   1:  PR[GP1:91,1] = PR[GP1:90,1] + 125.067;
   1:  PR[GP1:91,2] = PR[GP1:90,2] + 105.676;
   1:L PR[91] 10mm/sec FINE;
   1:  PR[GP1:91,1] = PR[GP1:90,1] + 125.211;
   1:  PR[GP1:91,2] = PR[GP1:90,2] + 108.371;
   1:L PR[91] 10mm/sec FINE;
   1:  PR[GP1:91,1] = PR[GP1:90,1] + 124.783;
   1:  PR[GP1:91,2] = PR[GP1:90,2] + 111.876;
   1:L PR[91] 10mm/sec FINE;
   1:  PR[GP1:91,1] = PR[GP1:90,1] + 123.660;
   1:  PR[GP1:91,2] = PR[GP1:90,2] + 115.178;
   1:L PR[91] 10mm/sec FINE;
   1:  PR[GP1:91,1] = PR[GP1:90,1] + 121.852;
   1:  PR[GP1:91,2] = PR[GP1:90,2] + 118.170;
   1:L PR[91] 10mm/sec FINE;
   1:  PR[GP1:91,1] = PR[GP1:90,1] + 119.446;
   1:  PR[GP1:91,2] = PR[GP1:90,2] + 120.740;
   1:L PR[91] 10mm/sec FINE;
   1:  PR[GP1:91,1] = PR[GP1:90,1] + 116.594;
   1:  PR[GP1:91,2] = PR[GP1:90,2] + 122.770;
   1:L PR[91] 10mm/sec FINE;
   1:  PR[GP1:91,1] = PR[GP1:90,1] + 113.357;
   1:  PR[GP1:91,2] = PR[GP1:90,2] + 124.215;
   1:L PR[91] 10mm/sec FINE;
   1:  PR[GP1:91,1] = PR[GP1:90,1] + 109.836;
   1:  PR[GP1:91,2] = PR[GP1:90,2] + 125.035;
   1:L PR[91] 10mm/sec FINE;
   1:  PR[GP1:91,1] = PR[GP1:90,1] + 106.255;
   1:  PR[GP1:91,2] = PR[GP1:90,2] + 125.172;
   1:L PR[91] 10mm/sec FINE;
   1:  PR[GP1:91,1] = PR[GP1:90,1] + 102.748;
   1:  PR[GP1:91,2] = PR[GP1:90,2] + 124.631;
   1:L PR[91] 10mm/sec FINE;
   1:  PR[GP1:91,1] = PR[GP1:90,1] + 99.339;
   1:  PR[GP1:91,2] = PR[GP1:90,2] + 123.456;
   1:L PR[91] 10mm/sec FINE;
   1:  PR[GP1:91,1] = PR[GP1:90,1] + 97.309;
   1:  PR[GP1:91,2] = PR[GP1:90,2] + 122.401;
   1:L PR[91] 10mm/sec FINE;
   1:  PR[GP1:91,1] = PR[GP1:90,1] + 96.953;
   1:  PR[GP1:91,2] = PR[GP1:90,2] + 122.201;
   1:L PR[91] 10mm/sec FINE;
   1:  PR[GP1:91,1] = PR[GP1:90,1] + 95.813;
   1:  PR[GP1:91,2] = PR[GP1:90,2] + 121.862;
   1:L PR[91] 10mm/sec FINE;
   1:  PR[GP1:91,1] = PR[GP1:90,1] + 94.847;
   1:  PR[GP1:91,2] = PR[GP1:90,2] + 122.067;
   1:L PR[91] 10mm/sec FINE;
   1:  PR[GP1:91,1] = PR[GP1:90,1] + 93.928;
   1:  PR[GP1:91,2] = PR[GP1:90,2] + 122.476;
   1:L PR[91] 10mm/sec FINE;
   1:  PR[GP1:91,1] = PR[GP1:90,1] + 93.286;
   1:  PR[GP1:91,2] = PR[GP1:90,2] + 122.743;
   1:L PR[91] 10mm/sec FINE;
   1:  PR[GP1:91,1] = PR[GP1:90,1] + 90.578;
   1:  PR[GP1:91,2] = PR[GP1:90,2] + 123.691;
   1:L PR[91] 10mm/sec FINE;
   1:  PR[GP1:91,1] = PR[GP1:90,1] + 89.346;
   1:  PR[GP1:91,2] = PR[GP1:90,2] + 123.990;
   1:L PR[91] 10mm/sec FINE;
   1:  PR[GP1:91,1] = PR[GP1:90,1] + 87.282;
   1:  PR[GP1:91,2] = PR[GP1:90,2] + 124.465;
   1:L PR[91] 10mm/sec FINE;
   1:  PR[GP1:91,1] = PR[GP1:90,1] + 86.381;
   1:  PR[GP1:91,2] = PR[GP1:90,2] + 124.569;
   1:L PR[91] 10mm/sec FINE;
   1:  PR[GP1:91,1] = PR[GP1:90,1] + 83.107;
   1:  PR[GP1:91,2] = PR[GP1:90,2] + 124.845;
   1:L PR[91] 10mm/sec FINE;
   1:  PR[GP1:91,1] = PR[GP1:90,1] + 82.927;
   1:  PR[GP1:91,2] = PR[GP1:90,2] + 124.844;
   1:L PR[91] 10mm/sec FINE;
   1:  PR[GP1:91,1] = PR[GP1:90,1] + 79.793;
   1:  PR[GP1:91,2] = PR[GP1:90,2] + 124.596;
   1:L PR[91] 10mm/sec FINE;
   1:  PR[GP1:91,1] = PR[GP1:90,1] + 78.215;
   1:  PR[GP1:91,2] = PR[GP1:90,2] + 124.296;
   1:L PR[91] 10mm/sec FINE;
   1:  PR[GP1:91,1] = PR[GP1:90,1] + 76.415;
   1:  PR[GP1:91,2] = PR[GP1:90,2] + 123.822;
   1:L PR[91] 10mm/sec FINE;
   1:  PR[GP1:91,1] = PR[GP1:90,1] + 73.897;
   1:  PR[GP1:91,2] = PR[GP1:90,2] + 122.815;
   1:L PR[91] 10mm/sec FINE;
   1:  PR[GP1:91,1] = PR[GP1:90,1] + 73.134;
   1:  PR[GP1:91,2] = PR[GP1:90,2] + 122.451;
   1:L PR[91] 10mm/sec FINE;
   1:  PR[GP1:91,1] = PR[GP1:90,1] + 70.131;
   1:  PR[GP1:91,2] = PR[GP1:90,2] + 120.456;
   1:L PR[91] 10mm/sec FINE;
   1:  PR[GP1:91,1] = PR[GP1:90,1] + 69.386;
   1:  PR[GP1:91,2] = PR[GP1:90,2] + 119.681;
   1:L PR[91] 10mm/sec FINE;
   1:  PR[GP1:91,1] = PR[GP1:90,1] + 67.649;
   1:  PR[GP1:91,2] = PR[GP1:90,2] + 117.796;
   1:L PR[91] 10mm/sec FINE;
   1:  PR[GP1:91,1] = PR[GP1:90,1] + 65.840;
   1:  PR[GP1:91,2] = PR[GP1:90,2] + 114.671;
   1:L PR[91] 10mm/sec FINE;
   1:  PR[GP1:91,1] = PR[GP1:90,1] + 64.732;
   1:  PR[GP1:91,2] = PR[GP1:90,2] + 111.266;
   1:L PR[91] 10mm/sec FINE;
   1:  PR[GP1:91,1] = PR[GP1:90,1] + 64.492;
   1:  PR[GP1:91,2] = PR[GP1:90,2] + 107.656;
   1:L PR[91] 10mm/sec FINE;
   1:  PR[GP1:91,1] = PR[GP1:90,1] + 65.074;
   1:  PR[GP1:91,2] = PR[GP1:90,2] + 104.024;
   1:L PR[91] 10mm/sec FINE;
   1:  PR[GP1:91,1] = PR[GP1:90,1] + 65.085;
   1:  PR[GP1:91,2] = PR[GP1:90,2] + 103.970;
   1:L PR[91] 10mm/sec FINE;
   1:  PR[GP1:91,1] = PR[GP1:90,1] + 66.507;
   1:  PR[GP1:91,2] = PR[GP1:90,2] + 100.470;
   1:L PR[91] 10mm/sec FINE;
   1:  PR[GP1:91,1] = PR[GP1:90,1] + 66.955;
   1:  PR[GP1:91,2] = PR[GP1:90,2] + 99.803;
   1:L PR[91] 10mm/sec FINE;
   1:  PR[GP1:91,1] = PR[GP1:90,1] + 68.693;
   1:  PR[GP1:91,2] = PR[GP1:90,2] + 97.301;
   1:L PR[91] 10mm/sec FINE;
   1:  PR[GP1:91,1] = PR[GP1:90,1] + 70.114;
   1:  PR[GP1:91,2] = PR[GP1:90,2] + 95.877;
   1:L PR[91] 10mm/sec FINE;
   1:  PR[GP1:91,1] = PR[GP1:90,1] + 71.437;
   1:  PR[GP1:91,2] = PR[GP1:90,2] + 94.608;
   1:L PR[91] 10mm/sec FINE;
   1:  PR[GP1:91,1] = PR[GP1:90,1] + 73.564;
   1:  PR[GP1:91,2] = PR[GP1:90,2] + 93.370;
   1:  PR[GP1:91,3] = PR[GP1:90,3] + 32.900;
   1:L PR[91] 10mm/sec FINE;
   1:  PR[GP1:91,1] = PR[GP1:90,1] + 75.182;
   1:  PR[GP1:91,2] = PR[GP1:90,2] + 92.299;
   1:L PR[91] 10mm/sec FINE;
   1:  PR[GP1:91,1] = PR[GP1:90,1] + 76.014;
   1:  PR[GP1:91,2] = PR[GP1:90,2] + 91.905;
   1:L PR[91] 10mm/sec FINE;
   1:  PR[GP1:91,1] = PR[GP1:90,1] + 78.652;
   1:  PR[GP1:91,2] = PR[GP1:90,2] + 90.708;
   1:L PR[91] 10mm/sec FINE;
   1:  PR[GP1:91,1] = PR[GP1:90,1] + 81.260;
   1:  PR[GP1:91,2] = PR[GP1:90,2] + 89.873;
   1:L PR[91] 10mm/sec FINE;
   1:  PR[GP1:91,1] = PR[GP1:90,1] + 81.725;
   1:  PR[GP1:91,2] = PR[GP1:90,2] + 89.744;
   1:L PR[91] 10mm/sec FINE;
   1:  PR[GP1:91,1] = PR[GP1:90,1] + 82.381;
   1:  PR[GP1:91,2] = PR[GP1:90,2] + 89.624;
   1:L PR[91] 10mm/sec FINE;
   1:  PR[GP1:91,1] = PR[GP1:90,1] + 85.201;
   1:  PR[GP1:91,2] = PR[GP1:90,2] + 89.020;
   1:L PR[91] 10mm/sec FINE;
   1:  PR[GP1:91,1] = PR[GP1:90,1] + 87.810;
   1:  PR[GP1:91,2] = PR[GP1:90,2] + 88.790;
   1:L PR[91] 10mm/sec FINE;
   1:  PR[GP1:91,1] = PR[GP1:90,1] + 89.579;
   1:  PR[GP1:91,2] = PR[GP1:90,2] + 88.697;
   1:L PR[91] 10mm/sec FINE;
   1:  PR[GP1:91,1] = PR[GP1:90,1] + 91.610;
   1:  PR[GP1:91,2] = PR[GP1:90,2] + 88.771;
   1:L PR[91] 10mm/sec FINE;
   1:  PR[GP1:91,1] = PR[GP1:90,1] + 94.675;
   1:  PR[GP1:91,2] = PR[GP1:90,2] + 89.210;
   1:L PR[91] 10mm/sec FINE;
   1:  PR[GP1:91,1] = PR[GP1:90,1] + 95.921;
   1:  PR[GP1:91,2] = PR[GP1:90,2] + 89.430;
   1:L PR[91] 10mm/sec FINE;
   1:  PR[GP1:91,1] = PR[GP1:90,1] + 97.181;
   1:  PR[GP1:91,2] = PR[GP1:90,2] + 89.860;
   1:L PR[91] 10mm/sec FINE;
   1:  PR[GP1:91,1] = PR[GP1:90,1] + 97.451;
   1:  PR[GP1:91,2] = PR[GP1:90,2] + 89.925;
   1:L PR[91] 10mm/sec FINE;
   1:  PR[GP1:91,1] = PR[GP1:90,1] + 98.662;
   1:  PR[GP1:91,2] = PR[GP1:90,2] + 89.766;
   1:L PR[91] 10mm/sec FINE;
   1:  PR[GP1:91,1] = PR[GP1:90,1] + 100.674;
   1:  PR[GP1:91,2] = PR[GP1:90,2] + 89.073;
   1:L PR[91] 10mm/sec FINE;
   1:  PR[GP1:91,1] = PR[GP1:90,1] + 100.904;
   1:  PR[GP1:91,2] = PR[GP1:90,2] + 88.999;
   1:L PR[91] 10mm/sec FINE;
   1:  PR[GP1:91,1] = PR[GP1:90,1] + 101.374;
   1:  PR[GP1:91,2] = PR[GP1:90,2] + 88.890;
   1:L PR[91] 10mm/sec FINE;
   1:  PR[GP1:91,1] = PR[GP1:90,1] + 103.724;
   1:  PR[GP1:91,2] = PR[GP1:90,2] + 88.477;
   1:L PR[91] 10mm/sec FINE;
   1:  PR[GP1:91,1] = PR[GP1:90,1] + 104.087;
   1:  PR[GP1:91,2] = PR[GP1:90,2] + 88.454;
   1:L PR[91] 10mm/sec FINE;
   1:  PR[GP1:91,1] = PR[GP1:90,1] + 106.621;
   1:  PR[GP1:91,2] = PR[GP1:90,2] + 88.429;
   1:L PR[91] 10mm/sec FINE;
   1:  PR[GP1:91,1] = PR[GP1:90,1] + 109.525;
   1:  PR[GP1:91,2] = PR[GP1:90,2] + 88.858;
   1:L PR[91] 10mm/sec FINE;
   1:  PR[GP1:91,1] = PR[GP1:90,1] + 112.350;
   1:  PR[GP1:91,2] = PR[GP1:90,2] + 89.744;
   1:L PR[91] 10mm/sec FINE;
   1:  PR[GP1:91,1] = PR[GP1:90,1] + 115.027;
   1:  PR[GP1:91,2] = PR[GP1:90,2] + 91.077;
   1:L PR[91] 10mm/sec FINE;
   1:  PR[GP1:91,1] = PR[GP1:90,1] + 117.480;
   1:  PR[GP1:91,2] = PR[GP1:90,2] + 92.827;
   1:L PR[91] 10mm/sec FINE;
   1:  PR[GP1:91,1] = PR[GP1:90,1] + 119.096;
   1:  PR[GP1:91,2] = PR[GP1:90,2] + 94.413;
   1:L PR[91] 10mm/sec FINE;
   1:  PR[GP1:91,1] = PR[GP1:90,1] + 119.702;
   1:  PR[GP1:91,2] = PR[GP1:90,2] + 94.984;
   1:L PR[91] 10mm/sec FINE;
   1:  PR[GP1:91,1] = PR[GP1:90,1] + 121.111;
   1:  PR[GP1:91,2] = PR[GP1:90,2] + 96.735;
   1:L PR[91] 10mm/sec FINE;
   1:  PR[GP1:91,1] = PR[GP1:90,1] + 121.662;
   1:  PR[GP1:91,2] = PR[GP1:90,2] + 97.494;
   1:L PR[91] 10mm/sec FINE;
   1:  PR[GP1:91,1] = PR[GP1:90,1] + 122.375;
   1:  PR[GP1:91,2] = PR[GP1:90,2] + 98.721;
   1:L PR[91] 10mm/sec FINE;
   1:  PR[GP1:91,1] = PR[GP1:90,1] + 123.132;
   1:  PR[GP1:91,2] = PR[GP1:90,2] + 100.157;
   1:L PR[91] 10mm/sec FINE;
   1:  PR[GP1:91,1] = PR[GP1:90,1] + 123.382;
   1:  PR[GP1:91,2] = PR[GP1:90,2] + 100.787;
   1:L PR[91] 10mm/sec FINE;
   1:  PR[GP1:91,1] = PR[GP1:90,1] + 124.131;
   1:  PR[GP1:91,2] = PR[GP1:90,2] + 102.876;
   1:L PR[91] 10mm/sec FINE;
   1:  PR[GP1:91,1] = PR[GP1:90,1] + 124.717;
   1:  PR[GP1:91,2] = PR[GP1:90,2] + 105.523;
   1:L PR[91] 10mm/sec FINE;
   1:  PR[GP1:91,1] = PR[GP1:90,1] + 124.859;
   1:  PR[GP1:91,2] = PR[GP1:90,2] + 108.206;
   1:L PR[91] 10mm/sec FINE;
   1:  PR[GP1:91,1] = PR[GP1:90,1] + 124.427;
   1:  PR[GP1:91,2] = PR[GP1:90,2] + 111.723;
   1:L PR[91] 10mm/sec FINE;
   1:  PR[GP1:91,1] = PR[GP1:90,1] + 123.294;
   1:  PR[GP1:91,2] = PR[GP1:90,2] + 115.038;
   1:L PR[91] 10mm/sec FINE;
   1:  PR[GP1:91,1] = PR[GP1:90,1] + 121.502;
   1:  PR[GP1:91,2] = PR[GP1:90,2] + 118.026;
   1:L PR[91] 10mm/sec FINE;
   1:  PR[GP1:91,1] = PR[GP1:90,1] + 119.130;
   1:  PR[GP1:91,2] = PR[GP1:90,2] + 120.582;
   1:L PR[91] 10mm/sec FINE;
   1:  PR[GP1:91,1] = PR[GP1:90,1] + 118.062;
   1:  PR[GP1:91,2] = PR[GP1:90,2] + 121.345;
   1:L PR[91] 10mm/sec FINE;
   1:  PR[GP1:91,1] = PR[GP1:90,1] + 116.272;
   1:  PR[GP1:91,2] = PR[GP1:90,2] + 122.619;
   1:L PR[91] 10mm/sec FINE;
   1:  PR[GP1:91,1] = PR[GP1:90,1] + 113.025;
   1:  PR[GP1:91,2] = PR[GP1:90,2] + 124.072;
   1:L PR[91] 10mm/sec FINE;
   1:  PR[GP1:91,1] = PR[GP1:90,1] + 109.576;
   1:  PR[GP1:91,2] = PR[GP1:90,2] + 124.872;
   1:L PR[91] 10mm/sec FINE;
   1:  PR[GP1:91,1] = PR[GP1:90,1] + 106.003;
   1:  PR[GP1:91,2] = PR[GP1:90,2] + 125.012;
   1:L PR[91] 10mm/sec FINE;
   1:  PR[GP1:91,1] = PR[GP1:90,1] + 104.565;
   1:  PR[GP1:91,2] = PR[GP1:90,2] + 124.806;
   1:L PR[91] 10mm/sec FINE;
   1:  PR[GP1:91,1] = PR[GP1:90,1] + 102.475;
   1:  PR[GP1:91,2] = PR[GP1:90,2] + 124.481;
   1:L PR[91] 10mm/sec FINE;
   1:  PR[GP1:91,1] = PR[GP1:90,1] + 99.066;
   1:  PR[GP1:91,2] = PR[GP1:90,2] + 123.311;
   1:L PR[91] 10mm/sec FINE;
   1:  PR[GP1:91,1] = PR[GP1:90,1] + 97.099;
   1:  PR[GP1:91,2] = PR[GP1:90,2] + 122.284;
   1:L PR[91] 10mm/sec FINE;
   1:  PR[GP1:91,1] = PR[GP1:90,1] + 96.627;
   1:  PR[GP1:91,2] = PR[GP1:90,2] + 122.161;
   1:L PR[91] 10mm/sec FINE;
   1:  PR[GP1:91,1] = PR[GP1:90,1] + 95.962;
   1:  PR[GP1:91,2] = PR[GP1:90,2] + 121.960;
   1:L PR[91] 10mm/sec FINE;
   1:  PR[GP1:91,1] = PR[GP1:90,1] + 95.071;
   1:  PR[GP1:91,2] = PR[GP1:90,2] + 122.159;
   1:L PR[91] 10mm/sec FINE;
   1:  PR[GP1:91,1] = PR[GP1:90,1] + 93.990;
   1:  PR[GP1:91,2] = PR[GP1:90,2] + 122.603;
   1:L PR[91] 10mm/sec FINE;
   1:  PR[GP1:91,1] = PR[GP1:90,1] + 91.198;
   1:  PR[GP1:91,2] = PR[GP1:90,2] + 123.560;
   1:L PR[91] 10mm/sec FINE;
   1:  PR[GP1:91,1] = PR[GP1:90,1] + 88.055;
   1:  PR[GP1:91,2] = PR[GP1:90,2] + 124.289;
   1:L PR[91] 10mm/sec FINE;
   1:  PR[GP1:91,1] = PR[GP1:90,1] + 86.606;
   1:  PR[GP1:91,2] = PR[GP1:90,2] + 124.457;
   1:L PR[91] 10mm/sec FINE;
   1:  PR[GP1:91,1] = PR[GP1:90,1] + 83.984;
   1:  PR[GP1:91,2] = PR[GP1:90,2] + 124.674;
   1:L PR[91] 10mm/sec FINE;
   1:  PR[GP1:91,1] = PR[GP1:90,1] + 83.485;
   1:  PR[GP1:91,2] = PR[GP1:90,2] + 124.677;
   1:L PR[91] 10mm/sec FINE;
   1:  PR[GP1:91,1] = PR[GP1:90,1] + 80.051;
   1:  PR[GP1:91,2] = PR[GP1:90,2] + 124.408;
   1:L PR[91] 10mm/sec FINE;
   1:  PR[GP1:91,1] = PR[GP1:90,1] + 79.265;
   1:  PR[GP1:91,2] = PR[GP1:90,2] + 124.259;
   1:L PR[91] 10mm/sec FINE;
   1:  PR[GP1:91,1] = PR[GP1:90,1] + 76.736;
   1:  PR[GP1:91,2] = PR[GP1:90,2] + 123.592;
   1:L PR[91] 10mm/sec FINE;
   1:  PR[GP1:91,1] = PR[GP1:90,1] + 74.918;
   1:  PR[GP1:91,2] = PR[GP1:90,2] + 122.866;
   1:L PR[91] 10mm/sec FINE;
   1:  PR[GP1:91,1] = PR[GP1:90,1] + 73.515;
   1:  PR[GP1:91,2] = PR[GP1:90,2] + 122.198;
   1:L PR[91] 10mm/sec FINE;
   1:  PR[GP1:91,1] = PR[GP1:90,1] + 71.197;
   1:  PR[GP1:91,2] = PR[GP1:90,2] + 120.664;
   1:L PR[91] 10mm/sec FINE;
   1:  PR[GP1:91,1] = PR[GP1:90,1] + 70.574;
   1:  PR[GP1:91,2] = PR[GP1:90,2] + 120.197;
   1:L PR[91] 10mm/sec FINE;
   1:  PR[GP1:91,1] = PR[GP1:90,1] + 68.301;
   1:  PR[GP1:91,2] = PR[GP1:90,2] + 117.833;
   1:L PR[91] 10mm/sec FINE;
   1:  PR[GP1:91,1] = PR[GP1:90,1] + 68.113;
   1:  PR[GP1:91,2] = PR[GP1:90,2] + 117.615;
   1:L PR[91] 10mm/sec FINE;
   1:  PR[GP1:91,1] = PR[GP1:90,1] + 66.280;
   1:  PR[GP1:91,2] = PR[GP1:90,2] + 114.537;
   1:L PR[91] 10mm/sec FINE;
   1:  PR[GP1:91,1] = PR[GP1:90,1] + 65.163;
   1:  PR[GP1:91,2] = PR[GP1:90,2] + 111.135;
   1:L PR[91] 10mm/sec FINE;
   1:  PR[GP1:91,1] = PR[GP1:90,1] + 64.981;
   1:  PR[GP1:91,2] = PR[GP1:90,2] + 107.692;
   1:L PR[91] 10mm/sec FINE;
   1:  PR[GP1:91,1] = PR[GP1:90,1] + 64.960;
   1:  PR[GP1:91,2] = PR[GP1:90,2] + 107.499;
   1:L PR[91] 10mm/sec FINE;
   1:  PR[GP1:91,1] = PR[GP1:90,1] + 65.415;
   1:  PR[GP1:91,2] = PR[GP1:90,2] + 104.903;
   1:L PR[91] 10mm/sec FINE;
   1:  PR[GP1:91,1] = PR[GP1:90,1] + 65.548;
   1:  PR[GP1:91,2] = PR[GP1:90,2] + 104.351;
   1:L PR[91] 10mm/sec FINE;
   1:  PR[GP1:91,1] = PR[GP1:90,1] + 65.650;
   1:  PR[GP1:91,2] = PR[GP1:90,2] + 103.812;
   1:L PR[91] 10mm/sec FINE;
   1:  PR[GP1:91,1] = PR[GP1:90,1] + 67.051;
   1:  PR[GP1:91,2] = PR[GP1:90,2] + 100.343;
   1:L PR[91] 10mm/sec FINE;
   1:  PR[GP1:91,1] = PR[GP1:90,1] + 67.947;
   1:  PR[GP1:91,2] = PR[GP1:90,2] + 99.007;
   1:L PR[91] 10mm/sec FINE;
   1:  PR[GP1:91,1] = PR[GP1:90,1] + 69.205;
   1:  PR[GP1:91,2] = PR[GP1:90,2] + 97.197;
   1:L PR[91] 10mm/sec FINE;
   1:  PR[GP1:91,1] = PR[GP1:90,1] + 71.256;
   1:  PR[GP1:91,2] = PR[GP1:90,2] + 95.142;
   1:L PR[91] 10mm/sec FINE;
   1:  PR[GP1:91,1] = PR[GP1:90,1] + 71.906;
   1:  PR[GP1:91,2] = PR[GP1:90,2] + 94.518;
   1:L PR[91] 10mm/sec FINE;
   1:  PR[GP1:91,1] = PR[GP1:90,1] + 75.880;
   1:  PR[GP1:91,2] = PR[GP1:90,2] + 92.109;
   1:  PR[GP1:91,3] = PR[GP1:90,3] + 33.900;
   1:L PR[91] 10mm/sec FINE;
   1:  PR[GP1:91,1] = PR[GP1:90,1] + 77.710;
   1:  PR[GP1:91,2] = PR[GP1:90,2] + 91.243;
   1:L PR[91] 10mm/sec FINE;
   1:  PR[GP1:91,1] = PR[GP1:90,1] + 79.190;
   1:  PR[GP1:91,2] = PR[GP1:90,2] + 90.572;
   1:L PR[91] 10mm/sec FINE;
   1:  PR[GP1:91,1] = PR[GP1:90,1] + 81.284;
   1:  PR[GP1:91,2] = PR[GP1:90,2] + 89.901;
   1:L PR[91] 10mm/sec FINE;
   1:  PR[GP1:91,1] = PR[GP1:90,1] + 82.269;
   1:  PR[GP1:91,2] = PR[GP1:90,2] + 89.559;
   1:L PR[91] 10mm/sec FINE;
   1:  PR[GP1:91,1] = PR[GP1:90,1] + 86.037;
   1:  PR[GP1:91,2] = PR[GP1:90,2] + 88.743;
   1:L PR[91] 10mm/sec FINE;
   1:  PR[GP1:91,1] = PR[GP1:90,1] + 88.313;
   1:  PR[GP1:91,2] = PR[GP1:90,2] + 88.542;
   1:L PR[91] 10mm/sec FINE;
   1:  PR[GP1:91,1] = PR[GP1:90,1] + 90.636;
   1:  PR[GP1:91,2] = PR[GP1:90,2] + 88.420;
   1:L PR[91] 10mm/sec FINE;
   1:  PR[GP1:91,1] = PR[GP1:90,1] + 92.273;
   1:  PR[GP1:91,2] = PR[GP1:90,2] + 88.479;
   1:L PR[91] 10mm/sec FINE;
   1:  PR[GP1:91,1] = PR[GP1:90,1] + 95.963;
   1:  PR[GP1:91,2] = PR[GP1:90,2] + 89.008;
   1:L PR[91] 10mm/sec FINE;
   1:  PR[GP1:91,1] = PR[GP1:90,1] + 96.765;
   1:  PR[GP1:91,2] = PR[GP1:90,2] + 89.149;
   1:L PR[91] 10mm/sec FINE;
   1:  PR[GP1:91,1] = PR[GP1:90,1] + 97.566;
   1:  PR[GP1:91,2] = PR[GP1:90,2] + 89.421;
   1:L PR[91] 10mm/sec FINE;
   1:  PR[GP1:91,1] = PR[GP1:90,1] + 97.747;
   1:  PR[GP1:91,2] = PR[GP1:90,2] + 89.464;
   1:L PR[91] 10mm/sec FINE;
   1:  PR[GP1:91,1] = PR[GP1:90,1] + 98.964;
   1:  PR[GP1:91,2] = PR[GP1:90,2] + 89.336;
   1:L PR[91] 10mm/sec FINE;
   1:  PR[GP1:91,1] = PR[GP1:90,1] + 100.640;
   1:  PR[GP1:91,2] = PR[GP1:90,2] + 88.779;
   1:L PR[91] 10mm/sec FINE;
   1:  PR[GP1:91,1] = PR[GP1:90,1] + 101.756;
   1:  PR[GP1:91,2] = PR[GP1:90,2] + 88.520;
   1:L PR[91] 10mm/sec FINE;
   1:  PR[GP1:91,1] = PR[GP1:90,1] + 103.448;
   1:  PR[GP1:91,2] = PR[GP1:90,2] + 88.222;
   1:L PR[91] 10mm/sec FINE;
   1:  PR[GP1:91,1] = PR[GP1:90,1] + 104.526;
   1:  PR[GP1:91,2] = PR[GP1:90,2] + 88.154;
   1:L PR[91] 10mm/sec FINE;
   1:  PR[GP1:91,1] = PR[GP1:90,1] + 106.342;
   1:  PR[GP1:91,2] = PR[GP1:90,2] + 88.137;
   1:L PR[91] 10mm/sec FINE;
   1:  PR[GP1:91,1] = PR[GP1:90,1] + 107.253;
   1:  PR[GP1:91,2] = PR[GP1:90,2] + 88.230;
   1:L PR[91] 10mm/sec FINE;
   1:  PR[GP1:91,1] = PR[GP1:90,1] + 109.250;
   1:  PR[GP1:91,2] = PR[GP1:90,2] + 88.541;
   1:L PR[91] 10mm/sec FINE;
   1:  PR[GP1:91,1] = PR[GP1:90,1] + 109.859;
   1:  PR[GP1:91,2] = PR[GP1:90,2] + 88.707;
   1:L PR[91] 10mm/sec FINE;
   1:  PR[GP1:91,1] = PR[GP1:90,1] + 112.092;
   1:  PR[GP1:91,2] = PR[GP1:90,2] + 89.441;
   1:L PR[91] 10mm/sec FINE;
   1:  PR[GP1:91,1] = PR[GP1:90,1] + 112.281;
   1:  PR[GP1:91,2] = PR[GP1:90,2] + 89.527;
   1:L PR[91] 10mm/sec FINE;
   1:  PR[GP1:91,1] = PR[GP1:90,1] + 113.192;
   1:  PR[GP1:91,2] = PR[GP1:90,2] + 90.000;
   1:L PR[91] 10mm/sec FINE;
   1:  PR[GP1:91,1] = PR[GP1:90,1] + 114.777;
   1:  PR[GP1:91,2] = PR[GP1:90,2] + 90.781;
   1:L PR[91] 10mm/sec FINE;
   1:  PR[GP1:91,1] = PR[GP1:90,1] + 117.237;
   1:  PR[GP1:91,2] = PR[GP1:90,2] + 92.516;
   1:L PR[91] 10mm/sec FINE;
   1:  PR[GP1:91,1] = PR[GP1:90,1] + 119.406;
   1:  PR[GP1:91,2] = PR[GP1:90,2] + 94.623;
   1:L PR[91] 10mm/sec FINE;
   1:  PR[GP1:91,1] = PR[GP1:90,1] + 121.236;
   1:  PR[GP1:91,2] = PR[GP1:90,2] + 97.056;
   1:L PR[91] 10mm/sec FINE;
   1:  PR[GP1:91,1] = PR[GP1:90,1] + 122.420;
   1:  PR[GP1:91,2] = PR[GP1:90,2] + 99.091;
   1:L PR[91] 10mm/sec FINE;
   1:  PR[GP1:91,1] = PR[GP1:90,1] + 122.771;
   1:  PR[GP1:91,2] = PR[GP1:90,2] + 99.758;
   1:L PR[91] 10mm/sec FINE;
   1:  PR[GP1:91,1] = PR[GP1:90,1] + 123.359;
   1:  PR[GP1:91,2] = PR[GP1:90,2] + 101.242;
   1:L PR[91] 10mm/sec FINE;
   1:  PR[GP1:91,1] = PR[GP1:90,1] + 123.821;
   1:  PR[GP1:91,2] = PR[GP1:90,2] + 102.530;
   1:L PR[91] 10mm/sec FINE;
   1:  PR[GP1:91,1] = PR[GP1:90,1] + 124.030;
   1:  PR[GP1:91,2] = PR[GP1:90,2] + 103.454;
   1:L PR[91] 10mm/sec FINE;
   1:  PR[GP1:91,1] = PR[GP1:90,1] + 124.403;
   1:  PR[GP1:91,2] = PR[GP1:90,2] + 105.299;
   1:L PR[91] 10mm/sec FINE;
   1:  PR[GP1:91,1] = PR[GP1:90,1] + 124.528;
   1:  PR[GP1:91,2] = PR[GP1:90,2] + 108.026;
   1:L PR[91] 10mm/sec FINE;
   1:  PR[GP1:91,1] = PR[GP1:90,1] + 124.113;
   1:  PR[GP1:91,2] = PR[GP1:90,2] + 111.543;
   1:L PR[91] 10mm/sec FINE;
   1:  PR[GP1:91,1] = PR[GP1:90,1] + 122.985;
   1:  PR[GP1:91,2] = PR[GP1:90,2] + 114.864;
   1:L PR[91] 10mm/sec FINE;
   1:  PR[GP1:91,1] = PR[GP1:90,1] + 121.192;
   1:  PR[GP1:91,2] = PR[GP1:90,2] + 117.859;
   1:L PR[91] 10mm/sec FINE;
   1:  PR[GP1:91,1] = PR[GP1:90,1] + 118.815;
   1:  PR[GP1:91,2] = PR[GP1:90,2] + 120.424;
   1:L PR[91] 10mm/sec FINE;
   1:  PR[GP1:91,1] = PR[GP1:90,1] + 115.950;
   1:  PR[GP1:91,2] = PR[GP1:90,2] + 122.468;
   1:L PR[91] 10mm/sec FINE;
   1:  PR[GP1:91,1] = PR[GP1:90,1] + 112.721;
   1:  PR[GP1:91,2] = PR[GP1:90,2] + 123.919;
   1:L PR[91] 10mm/sec FINE;
   1:  PR[GP1:91,1] = PR[GP1:90,1] + 109.316;
   1:  PR[GP1:91,2] = PR[GP1:90,2] + 124.709;
   1:L PR[91] 10mm/sec FINE;
   1:  PR[GP1:91,1] = PR[GP1:90,1] + 105.778;
   1:  PR[GP1:91,2] = PR[GP1:90,2] + 124.846;
   1:L PR[91] 10mm/sec FINE;
   1:  PR[GP1:91,1] = PR[GP1:90,1] + 102.203;
   1:  PR[GP1:91,2] = PR[GP1:90,2] + 124.331;
   1:L PR[91] 10mm/sec FINE;
   1:  PR[GP1:91,1] = PR[GP1:90,1] + 98.768;
   1:  PR[GP1:91,2] = PR[GP1:90,2] + 123.112;
   1:L PR[91] 10mm/sec FINE;
   1:  PR[GP1:91,1] = PR[GP1:90,1] + 98.344;
   1:  PR[GP1:91,2] = PR[GP1:90,2] + 122.907;
   1:L PR[91] 10mm/sec FINE;
   1:  PR[GP1:91,1] = PR[GP1:90,1] + 97.258;
   1:  PR[GP1:91,2] = PR[GP1:90,2] + 122.346;
   1:L PR[91] 10mm/sec FINE;
   1:  PR[GP1:91,1] = PR[GP1:90,1] + 96.108;
   1:  PR[GP1:91,2] = PR[GP1:90,2] + 122.055;
   1:L PR[91] 10mm/sec FINE;
   1:  PR[GP1:91,1] = PR[GP1:90,1] + 95.302;
   1:  PR[GP1:91,2] = PR[GP1:90,2] + 122.227;
   1:L PR[91] 10mm/sec FINE;
   1:  PR[GP1:91,1] = PR[GP1:90,1] + 94.695;
   1:  PR[GP1:91,2] = PR[GP1:90,2] + 122.463;
   1:L PR[91] 10mm/sec FINE;
   1:  PR[GP1:91,1] = PR[GP1:90,1] + 92.033;
   1:  PR[GP1:91,2] = PR[GP1:90,2] + 123.359;
   1:L PR[91] 10mm/sec FINE;
   1:  PR[GP1:91,1] = PR[GP1:90,1] + 88.828;
   1:  PR[GP1:91,2] = PR[GP1:90,2] + 124.113;
   1:L PR[91] 10mm/sec FINE;
   1:  PR[GP1:91,1] = PR[GP1:90,1] + 86.830;
   1:  PR[GP1:91,2] = PR[GP1:90,2] + 124.345;
   1:L PR[91] 10mm/sec FINE;
   1:  PR[GP1:91,1] = PR[GP1:90,1] + 85.063;
   1:  PR[GP1:91,2] = PR[GP1:90,2] + 124.491;
   1:L PR[91] 10mm/sec FINE;
   1:  PR[GP1:91,1] = PR[GP1:90,1] + 83.896;
   1:  PR[GP1:91,2] = PR[GP1:90,2] + 124.498;
   1:L PR[91] 10mm/sec FINE;
   1:  PR[GP1:91,1] = PR[GP1:90,1] + 80.317;
   1:  PR[GP1:91,2] = PR[GP1:90,2] + 124.221;
   1:L PR[91] 10mm/sec FINE;
   1:  PR[GP1:91,1] = PR[GP1:90,1] + 77.056;
   1:  PR[GP1:91,2] = PR[GP1:90,2] + 123.363;
   1:L PR[91] 10mm/sec FINE;
   1:  PR[GP1:91,1] = PR[GP1:90,1] + 75.938;
   1:  PR[GP1:91,2] = PR[GP1:90,2] + 122.916;
   1:L PR[91] 10mm/sec FINE;
   1:  PR[GP1:91,1] = PR[GP1:90,1] + 73.897;
   1:  PR[GP1:91,2] = PR[GP1:90,2] + 121.944;
   1:L PR[91] 10mm/sec FINE;
   1:  PR[GP1:91,1] = PR[GP1:90,1] + 72.163;
   1:  PR[GP1:91,2] = PR[GP1:90,2] + 120.797;
   1:L PR[91] 10mm/sec FINE;
   1:  PR[GP1:91,1] = PR[GP1:90,1] + 71.014;
   1:  PR[GP1:91,2] = PR[GP1:90,2] + 119.935;
   1:L PR[91] 10mm/sec FINE;
   1:  PR[GP1:91,1] = PR[GP1:90,1] + 69.191;
   1:  PR[GP1:91,2] = PR[GP1:90,2] + 118.039;
   1:L PR[91] 10mm/sec FINE;
   1:  PR[GP1:91,1] = PR[GP1:90,1] + 68.603;
   1:  PR[GP1:91,2] = PR[GP1:90,2] + 117.357;
   1:L PR[91] 10mm/sec FINE;
   1:  PR[GP1:91,1] = PR[GP1:90,1] + 67.108;
   1:  PR[GP1:91,2] = PR[GP1:90,2] + 114.852;
   1:L PR[91] 10mm/sec FINE;
   1:  PR[GP1:91,1] = PR[GP1:90,1] + 66.809;
   1:  PR[GP1:91,2] = PR[GP1:90,2] + 114.301;
   1:L PR[91] 10mm/sec FINE;
   1:  PR[GP1:91,1] = PR[GP1:90,1] + 65.875;
   1:  PR[GP1:91,2] = PR[GP1:90,2] + 111.457;
   1:L PR[91] 10mm/sec FINE;
   1:  PR[GP1:91,1] = PR[GP1:90,1] + 65.715;
   1:  PR[GP1:91,2] = PR[GP1:90,2] + 110.923;
   1:L PR[91] 10mm/sec FINE;
   1:  PR[GP1:91,1] = PR[GP1:90,1] + 65.562;
   1:  PR[GP1:91,2] = PR[GP1:90,2] + 108.031;
   1:L PR[91] 10mm/sec FINE;
   1:  PR[GP1:91,1] = PR[GP1:90,1] + 65.485;
   1:  PR[GP1:91,2] = PR[GP1:90,2] + 107.327;
   1:L PR[91] 10mm/sec FINE;
   1:  PR[GP1:91,1] = PR[GP1:90,1] + 65.756;
   1:  PR[GP1:91,2] = PR[GP1:90,2] + 105.779;
   1:L PR[91] 10mm/sec FINE;
   1:  PR[GP1:91,1] = PR[GP1:90,1] + 66.013;
   1:  PR[GP1:91,2] = PR[GP1:90,2] + 104.711;
   1:L PR[91] 10mm/sec FINE;
   1:  PR[GP1:91,1] = PR[GP1:90,1] + 66.214;
   1:  PR[GP1:91,2] = PR[GP1:90,2] + 103.656;
   1:L PR[91] 10mm/sec FINE;
   1:  PR[GP1:91,1] = PR[GP1:90,1] + 67.596;
   1:  PR[GP1:91,2] = PR[GP1:90,2] + 100.215;
   1:L PR[91] 10mm/sec FINE;
   1:  PR[GP1:91,1] = PR[GP1:90,1] + 68.940;
   1:  PR[GP1:91,2] = PR[GP1:90,2] + 98.212;
   1:L PR[91] 10mm/sec FINE;
   1:  PR[GP1:91,1] = PR[GP1:90,1] + 69.718;
   1:  PR[GP1:91,2] = PR[GP1:90,2] + 97.094;
   1:L PR[91] 10mm/sec FINE;
   1:  PR[GP1:91,1] = PR[GP1:90,1] + 72.381;
   1:  PR[GP1:91,2] = PR[GP1:90,2] + 94.425;
   1:L PR[91] 10mm/sec FINE;
   1:  PR[GP1:91,1] = PR[GP1:90,1] + 73.210;
   1:  PR[GP1:91,2] = PR[GP1:90,2] + 94.142;
   1:  PR[GP1:91,3] = PR[GP1:90,3] + 34.900;
   1:L PR[91] 10mm/sec FINE;
   1:  PR[GP1:91,1] = PR[GP1:90,1] + 75.364;
   1:  PR[GP1:91,2] = PR[GP1:90,2] + 92.708;
   1:L PR[91] 10mm/sec FINE;
   1:  PR[GP1:91,1] = PR[GP1:90,1] + 76.577;
   1:  PR[GP1:91,2] = PR[GP1:90,2] + 91.920;
   1:L PR[91] 10mm/sec FINE;
   1:  PR[GP1:91,1] = PR[GP1:90,1] + 79.728;
   1:  PR[GP1:91,2] = PR[GP1:90,2] + 90.435;
   1:L PR[91] 10mm/sec FINE;
   1:  PR[GP1:91,1] = PR[GP1:90,1] + 80.188;
   1:  PR[GP1:91,2] = PR[GP1:90,2] + 90.288;
   1:L PR[91] 10mm/sec FINE;
   1:  PR[GP1:91,1] = PR[GP1:90,1] + 82.928;
   1:  PR[GP1:91,2] = PR[GP1:90,2] + 89.336;
   1:L PR[91] 10mm/sec FINE;
   1:  PR[GP1:91,1] = PR[GP1:90,1] + 83.973;
   1:  PR[GP1:91,2] = PR[GP1:90,2] + 89.086;
   1:L PR[91] 10mm/sec FINE;
   1:  PR[GP1:91,1] = PR[GP1:90,1] + 86.873;
   1:  PR[GP1:91,2] = PR[GP1:90,2] + 88.465;
   1:L PR[91] 10mm/sec FINE;
   1:  PR[GP1:91,1] = PR[GP1:90,1] + 88.816;
   1:  PR[GP1:91,2] = PR[GP1:90,2] + 88.294;
   1:L PR[91] 10mm/sec FINE;
   1:  PR[GP1:91,1] = PR[GP1:90,1] + 91.692;
   1:  PR[GP1:91,2] = PR[GP1:90,2] + 88.143;
   1:L PR[91] 10mm/sec FINE;
   1:  PR[GP1:91,1] = PR[GP1:90,1] + 92.936;
   1:  PR[GP1:91,2] = PR[GP1:90,2] + 88.188;
   1:L PR[91] 10mm/sec FINE;
   1:  PR[GP1:91,1] = PR[GP1:90,1] + 97.250;
   1:  PR[GP1:91,2] = PR[GP1:90,2] + 88.806;
   1:L PR[91] 10mm/sec FINE;
   1:  PR[GP1:91,1] = PR[GP1:90,1] + 97.609;
   1:  PR[GP1:91,2] = PR[GP1:90,2] + 88.869;
   1:L PR[91] 10mm/sec FINE;
   1:  PR[GP1:91,1] = PR[GP1:90,1] + 98.056;
   1:  PR[GP1:91,2] = PR[GP1:90,2] + 89.015;
   1:L PR[91] 10mm/sec FINE;
   1:  PR[GP1:91,1] = PR[GP1:90,1] + 99.283;
   1:  PR[GP1:91,2] = PR[GP1:90,2] + 88.912;
   1:L PR[91] 10mm/sec FINE;
   1:  PR[GP1:91,1] = PR[GP1:90,1] + 100.374;
   1:  PR[GP1:91,2] = PR[GP1:90,2] + 88.560;
   1:L PR[91] 10mm/sec FINE;
   1:  PR[GP1:91,1] = PR[GP1:90,1] + 102.137;
   1:  PR[GP1:91,2] = PR[GP1:90,2] + 88.150;
   1:L PR[91] 10mm/sec FINE;
   1:  PR[GP1:91,1] = PR[GP1:90,1] + 103.172;
   1:  PR[GP1:91,2] = PR[GP1:90,2] + 87.968;
   1:L PR[91] 10mm/sec FINE;
   1:  PR[GP1:91,1] = PR[GP1:90,1] + 104.964;
   1:  PR[GP1:91,2] = PR[GP1:90,2] + 87.855;
   1:L PR[91] 10mm/sec FINE;
   1:  PR[GP1:91,1] = PR[GP1:90,1] + 106.059;
   1:  PR[GP1:91,2] = PR[GP1:90,2] + 87.844;
   1:L PR[91] 10mm/sec FINE;
   1:  PR[GP1:91,1] = PR[GP1:90,1] + 107.742;
   1:  PR[GP1:91,2] = PR[GP1:90,2] + 88.017;
   1:L PR[91] 10mm/sec FINE;
   1:  PR[GP1:91,1] = PR[GP1:90,1] + 108.966;
   1:  PR[GP1:91,2] = PR[GP1:90,2] + 88.207;
   1:L PR[91] 10mm/sec FINE;
   1:  PR[GP1:91,1] = PR[GP1:90,1] + 110.386;
   1:  PR[GP1:91,2] = PR[GP1:90,2] + 88.596;
   1:L PR[91] 10mm/sec FINE;
   1:  PR[GP1:91,1] = PR[GP1:90,1] + 111.814;
   1:  PR[GP1:91,2] = PR[GP1:90,2] + 89.065;
   1:L PR[91] 10mm/sec FINE;
   1:  PR[GP1:91,1] = PR[GP1:90,1] + 112.830;
   1:  PR[GP1:91,2] = PR[GP1:90,2] + 89.531;
   1:L PR[91] 10mm/sec FINE;
   1:  PR[GP1:91,1] = PR[GP1:90,1] + 114.519;
   1:  PR[GP1:91,2] = PR[GP1:90,2] + 90.407;
   1:L PR[91] 10mm/sec FINE;
   1:  PR[GP1:91,1] = PR[GP1:90,1] + 115.030;
   1:  PR[GP1:91,2] = PR[GP1:90,2] + 90.750;
   1:L PR[91] 10mm/sec FINE;
   1:  PR[GP1:91,1] = PR[GP1:90,1] + 116.992;
   1:  PR[GP1:91,2] = PR[GP1:90,2] + 92.202;
   1:L PR[91] 10mm/sec FINE;
   1:  PR[GP1:91,1] = PR[GP1:90,1] + 119.174;
   1:  PR[GP1:91,2] = PR[GP1:90,2] + 94.296;
   1:L PR[91] 10mm/sec FINE;
   1:  PR[GP1:91,1] = PR[GP1:90,1] + 121.000;
   1:  PR[GP1:91,2] = PR[GP1:90,2] + 96.706;
   1:L PR[91] 10mm/sec FINE;
   1:  PR[GP1:91,1] = PR[GP1:90,1] + 122.428;
   1:  PR[GP1:91,2] = PR[GP1:90,2] + 99.362;
   1:L PR[91] 10mm/sec FINE;
   1:  PR[GP1:91,1] = PR[GP1:90,1] + 122.585;
   1:  PR[GP1:91,2] = PR[GP1:90,2] + 99.801;
   1:L PR[91] 10mm/sec FINE;
   1:  PR[GP1:91,1] = PR[GP1:90,1] + 123.336;
   1:  PR[GP1:91,2] = PR[GP1:90,2] + 101.698;
   1:L PR[91] 10mm/sec FINE;
   1:  PR[GP1:91,1] = PR[GP1:90,1] + 123.510;
   1:  PR[GP1:91,2] = PR[GP1:90,2] + 102.183;
   1:L PR[91] 10mm/sec FINE;
   1:  PR[GP1:91,1] = PR[GP1:90,1] + 123.918;
   1:  PR[GP1:91,2] = PR[GP1:90,2] + 103.983;
   1:L PR[91] 10mm/sec FINE;
   1:  PR[GP1:91,1] = PR[GP1:90,1] + 124.125;
   1:  PR[GP1:91,2] = PR[GP1:90,2] + 105.009;
   1:L PR[91] 10mm/sec FINE;
   1:  PR[GP1:91,1] = PR[GP1:90,1] + 124.240;
   1:  PR[GP1:91,2] = PR[GP1:90,2] + 107.811;
   1:L PR[91] 10mm/sec FINE;
   1:  PR[GP1:91,1] = PR[GP1:90,1] + 123.799;
   1:  PR[GP1:91,2] = PR[GP1:90,2] + 111.361;
   1:L PR[91] 10mm/sec FINE;
   1:  PR[GP1:91,1] = PR[GP1:90,1] + 122.676;
   1:  PR[GP1:91,2] = PR[GP1:90,2] + 114.689;
   1:L PR[91] 10mm/sec FINE;
   1:  PR[GP1:91,1] = PR[GP1:90,1] + 120.881;
   1:  PR[GP1:91,2] = PR[GP1:90,2] + 117.693;
   1:L PR[91] 10mm/sec FINE;
   1:  PR[GP1:91,1] = PR[GP1:90,1] + 118.499;
   1:  PR[GP1:91,2] = PR[GP1:90,2] + 120.266;
   1:L PR[91] 10mm/sec FINE;
   1:  PR[GP1:91,1] = PR[GP1:90,1] + 115.648;
   1:  PR[GP1:91,2] = PR[GP1:90,2] + 122.310;
   1:L PR[91] 10mm/sec FINE;
   1:  PR[GP1:91,1] = PR[GP1:90,1] + 112.491;
   1:  PR[GP1:91,2] = PR[GP1:90,2] + 123.740;
   1:L PR[91] 10mm/sec FINE;
   1:  PR[GP1:91,1] = PR[GP1:90,1] + 109.055;
   1:  PR[GP1:91,2] = PR[GP1:90,2] + 124.546;
   1:L PR[91] 10mm/sec FINE;
   1:  PR[GP1:91,1] = PR[GP1:90,1] + 105.553;
   1:  PR[GP1:91,2] = PR[GP1:90,2] + 124.679;
   1:L PR[91] 10mm/sec FINE;
   1:  PR[GP1:91,1] = PR[GP1:90,1] + 103.066;
   1:  PR[GP1:91,2] = PR[GP1:90,2] + 124.323;
   1:L PR[91] 10mm/sec FINE;
   1:  PR[GP1:91,1] = PR[GP1:90,1] + 102.034;
   1:  PR[GP1:91,2] = PR[GP1:90,2] + 124.160;
   1:L PR[91] 10mm/sec FINE;
   1:  PR[GP1:91,1] = PR[GP1:90,1] + 98.706;
   1:  PR[GP1:91,2] = PR[GP1:90,2] + 122.981;
   1:L PR[91] 10mm/sec FINE;
   1:  PR[GP1:91,1] = PR[GP1:90,1] + 98.465;
   1:  PR[GP1:91,2] = PR[GP1:90,2] + 122.886;
   1:L PR[91] 10mm/sec FINE;
   1:  PR[GP1:91,1] = PR[GP1:90,1] + 97.422;
   1:  PR[GP1:91,2] = PR[GP1:90,2] + 122.385;
   1:L PR[91] 10mm/sec FINE;
   1:  PR[GP1:91,1] = PR[GP1:90,1] + 96.273;
   1:  PR[GP1:91,2] = PR[GP1:90,2] + 122.104;
   1:L PR[91] 10mm/sec FINE;
   1:  PR[GP1:91,1] = PR[GP1:90,1] + 95.542;
   1:  PR[GP1:91,2] = PR[GP1:90,2] + 122.269;
   1:L PR[91] 10mm/sec FINE;
   1:  PR[GP1:91,1] = PR[GP1:90,1] + 93.420;
   1:  PR[GP1:91,2] = PR[GP1:90,2] + 122.993;
   1:L PR[91] 10mm/sec FINE;
   1:  PR[GP1:91,1] = PR[GP1:90,1] + 92.912;
   1:  PR[GP1:91,2] = PR[GP1:90,2] + 123.145;
   1:L PR[91] 10mm/sec FINE;
   1:  PR[GP1:91,1] = PR[GP1:90,1] + 89.761;
   1:  PR[GP1:91,2] = PR[GP1:90,2] + 123.892;
   1:L PR[91] 10mm/sec FINE;
   1:  PR[GP1:91,1] = PR[GP1:90,1] + 88.560;
   1:  PR[GP1:91,2] = PR[GP1:90,2] + 124.057;
   1:L PR[91] 10mm/sec FINE;
   1:  PR[GP1:91,1] = PR[GP1:90,1] + 87.054;
   1:  PR[GP1:91,2] = PR[GP1:90,2] + 124.232;
   1:L PR[91] 10mm/sec FINE;
   1:  PR[GP1:91,1] = PR[GP1:90,1] + 86.143;
   1:  PR[GP1:91,2] = PR[GP1:90,2] + 124.308;
   1:L PR[91] 10mm/sec FINE;
   1:  PR[GP1:91,1] = PR[GP1:90,1] + 84.308;
   1:  PR[GP1:91,2] = PR[GP1:90,2] + 124.319;
   1:L PR[91] 10mm/sec FINE;
   1:  PR[GP1:91,1] = PR[GP1:90,1] + 81.691;
   1:  PR[GP1:91,2] = PR[GP1:90,2] + 124.117;
   1:L PR[91] 10mm/sec FINE;
   1:  PR[GP1:91,1] = PR[GP1:90,1] + 80.937;
   1:  PR[GP1:91,2] = PR[GP1:90,2] + 124.031;
   1:L PR[91] 10mm/sec FINE;
   1:  PR[GP1:91,1] = PR[GP1:90,1] + 78.637;
   1:  PR[GP1:91,2] = PR[GP1:90,2] + 123.466;
   1:L PR[91] 10mm/sec FINE;
   1:  PR[GP1:91,1] = PR[GP1:90,1] + 77.377;
   1:  PR[GP1:91,2] = PR[GP1:90,2] + 123.133;
   1:L PR[91] 10mm/sec FINE;
   1:  PR[GP1:91,1] = PR[GP1:90,1] + 76.959;
   1:  PR[GP1:91,2] = PR[GP1:90,2] + 122.966;
   1:L PR[91] 10mm/sec FINE;
   1:  PR[GP1:91,1] = PR[GP1:90,1] + 74.279;
   1:  PR[GP1:91,2] = PR[GP1:90,2] + 121.690;
   1:L PR[91] 10mm/sec FINE;
   1:  PR[GP1:91,1] = PR[GP1:90,1] + 73.130;
   1:  PR[GP1:91,2] = PR[GP1:90,2] + 120.930;
   1:L PR[91] 10mm/sec FINE;
   1:  PR[GP1:91,1] = PR[GP1:90,1] + 71.453;
   1:  PR[GP1:91,2] = PR[GP1:90,2] + 119.672;
   1:L PR[91] 10mm/sec FINE;
   1:  PR[GP1:91,1] = PR[GP1:90,1] + 70.081;
   1:  PR[GP1:91,2] = PR[GP1:90,2] + 118.246;
   1:L PR[91] 10mm/sec FINE;
   1:  PR[GP1:91,1] = PR[GP1:90,1] + 69.092;
   1:  PR[GP1:91,2] = PR[GP1:90,2] + 117.099;
   1:L PR[91] 10mm/sec FINE;
   1:  PR[GP1:91,1] = PR[GP1:90,1] + 67.910;
   1:  PR[GP1:91,2] = PR[GP1:90,2] + 115.118;
   1:L PR[91] 10mm/sec FINE;
   1:  PR[GP1:91,1] = PR[GP1:90,1] + 67.336;
   1:  PR[GP1:91,2] = PR[GP1:90,2] + 114.060;
   1:L PR[91] 10mm/sec FINE;
   1:  PR[GP1:91,1] = PR[GP1:90,1] + 66.583;
   1:  PR[GP1:91,2] = PR[GP1:90,2] + 111.766;
   1:L PR[91] 10mm/sec FINE;
   1:  PR[GP1:91,1] = PR[GP1:90,1] + 66.267;
   1:  PR[GP1:91,2] = PR[GP1:90,2] + 110.709;
   1:L PR[91] 10mm/sec FINE;
   1:  PR[GP1:91,1] = PR[GP1:90,1] + 66.143;
   1:  PR[GP1:91,2] = PR[GP1:90,2] + 108.371;
   1:L PR[91] 10mm/sec FINE;
   1:  PR[GP1:91,1] = PR[GP1:90,1] + 66.010;
   1:  PR[GP1:91,2] = PR[GP1:90,2] + 107.155;
   1:L PR[91] 10mm/sec FINE;
   1:  PR[GP1:91,1] = PR[GP1:90,1] + 66.097;
   1:  PR[GP1:91,2] = PR[GP1:90,2] + 106.655;
   1:L PR[91] 10mm/sec FINE;
   1:  PR[GP1:91,1] = PR[GP1:90,1] + 66.479;
   1:  PR[GP1:91,2] = PR[GP1:90,2] + 105.071;
   1:L PR[91] 10mm/sec FINE;
   1:  PR[GP1:91,1] = PR[GP1:90,1] + 66.778;
   1:  PR[GP1:91,2] = PR[GP1:90,2] + 103.500;
   1:L PR[91] 10mm/sec FINE;
   1:  PR[GP1:91,1] = PR[GP1:90,1] + 68.140;
   1:  PR[GP1:91,2] = PR[GP1:90,2] + 100.088;
   1:L PR[91] 10mm/sec FINE;
   1:  PR[GP1:91,1] = PR[GP1:90,1] + 70.231;
   1:  PR[GP1:91,2] = PR[GP1:90,2] + 96.989;
   1:L PR[91] 10mm/sec FINE;
   1:  PR[GP1:91,1] = PR[GP1:90,1] + 71.254;
   1:  PR[GP1:91,2] = PR[GP1:90,2] + 95.963;
   1:L PR[91] 10mm/sec FINE;
   1:  PR[GP1:91,1] = PR[GP1:90,1] + 72.787;
   1:  PR[GP1:91,2] = PR[GP1:90,2] + 94.504;
   1:L PR[91] 10mm/sec FINE;
   1:  PR[GP1:91,1] = PR[GP1:90,1] + 74.046;
   1:  PR[GP1:91,2] = PR[GP1:90,2] + 93.854;
   1:  PR[GP1:91,3] = PR[GP1:90,3] + 35.900;
   1:L PR[91] 10mm/sec FINE;
   1:  PR[GP1:91,1] = PR[GP1:90,1] + 75.631;
   1:  PR[GP1:91,2] = PR[GP1:90,2] + 92.799;
   1:L PR[91] 10mm/sec FINE;
   1:  PR[GP1:91,1] = PR[GP1:90,1] + 77.276;
   1:  PR[GP1:91,2] = PR[GP1:90,2] + 91.730;
   1:L PR[91] 10mm/sec FINE;
   1:  PR[GP1:91,1] = PR[GP1:90,1] + 80.270;
   1:  PR[GP1:91,2] = PR[GP1:90,2] + 90.298;
   1:L PR[91] 10mm/sec FINE;
   1:  PR[GP1:91,1] = PR[GP1:90,1] + 80.626;
   1:  PR[GP1:91,2] = PR[GP1:90,2] + 90.142;
   1:L PR[91] 10mm/sec FINE;
   1:  PR[GP1:91,1] = PR[GP1:90,1] + 83.586;
   1:  PR[GP1:91,2] = PR[GP1:90,2] + 89.114;
   1:L PR[91] 10mm/sec FINE;
   1:  PR[GP1:91,1] = PR[GP1:90,1] + 85.305;
   1:  PR[GP1:91,2] = PR[GP1:90,2] + 88.703;
   1:L PR[91] 10mm/sec FINE;
   1:  PR[GP1:91,1] = PR[GP1:90,1] + 87.709;
   1:  PR[GP1:91,2] = PR[GP1:90,2] + 88.188;
   1:L PR[91] 10mm/sec FINE;
   1:  PR[GP1:91,1] = PR[GP1:90,1] + 89.319;
   1:  PR[GP1:91,2] = PR[GP1:90,2] + 88.046;
   1:L PR[91] 10mm/sec FINE;
   1:  PR[GP1:91,1] = PR[GP1:90,1] + 92.748;
   1:  PR[GP1:91,2] = PR[GP1:90,2] + 87.866;
   1:L PR[91] 10mm/sec FINE;
   1:  PR[GP1:91,1] = PR[GP1:90,1] + 93.598;
   1:  PR[GP1:91,2] = PR[GP1:90,2] + 87.897;
   1:L PR[91] 10mm/sec FINE;
   1:  PR[GP1:91,1] = PR[GP1:90,1] + 98.131;
   1:  PR[GP1:91,2] = PR[GP1:90,2] + 88.546;
   1:L PR[91] 10mm/sec FINE;
   1:  PR[GP1:91,1] = PR[GP1:90,1] + 98.433;
   1:  PR[GP1:91,2] = PR[GP1:90,2] + 88.573;
   1:L PR[91] 10mm/sec FINE;
   1:  PR[GP1:91,1] = PR[GP1:90,1] + 99.618;
   1:  PR[GP1:91,2] = PR[GP1:90,2] + 88.495;
   1:L PR[91] 10mm/sec FINE;
   1:  PR[GP1:91,1] = PR[GP1:90,1] + 100.108;
   1:  PR[GP1:91,2] = PR[GP1:90,2] + 88.341;
   1:L PR[91] 10mm/sec FINE;
   1:  PR[GP1:91,1] = PR[GP1:90,1] + 102.519;
   1:  PR[GP1:91,2] = PR[GP1:90,2] + 87.780;
   1:L PR[91] 10mm/sec FINE;
   1:  PR[GP1:91,1] = PR[GP1:90,1] + 102.896;
   1:  PR[GP1:91,2] = PR[GP1:90,2] + 87.713;
   1:L PR[91] 10mm/sec FINE;
   1:  PR[GP1:91,1] = PR[GP1:90,1] + 105.403;
   1:  PR[GP1:91,2] = PR[GP1:90,2] + 87.555;
   1:L PR[91] 10mm/sec FINE;
   1:  PR[GP1:91,1] = PR[GP1:90,1] + 105.776;
   1:  PR[GP1:91,2] = PR[GP1:90,2] + 87.552;
   1:L PR[91] 10mm/sec FINE;
   1:  PR[GP1:91,1] = PR[GP1:90,1] + 108.230;
   1:  PR[GP1:91,2] = PR[GP1:90,2] + 87.804;
   1:L PR[91] 10mm/sec FINE;
   1:  PR[GP1:91,1] = PR[GP1:90,1] + 108.681;
   1:  PR[GP1:91,2] = PR[GP1:90,2] + 87.874;
   1:L PR[91] 10mm/sec FINE;
   1:  PR[GP1:91,1] = PR[GP1:90,1] + 110.913;
   1:  PR[GP1:91,2] = PR[GP1:90,2] + 88.485;
   1:L PR[91] 10mm/sec FINE;
   1:  PR[GP1:91,1] = PR[GP1:90,1] + 111.536;
   1:  PR[GP1:91,2] = PR[GP1:90,2] + 88.689;
   1:L PR[91] 10mm/sec FINE;
   1:  PR[GP1:91,1] = PR[GP1:90,1] + 113.380;
   1:  PR[GP1:91,2] = PR[GP1:90,2] + 89.534;
   1:L PR[91] 10mm/sec FINE;
   1:  PR[GP1:91,1] = PR[GP1:90,1] + 114.257;
   1:  PR[GP1:91,2] = PR[GP1:90,2] + 89.989;
   1:L PR[91] 10mm/sec FINE;
   1:  PR[GP1:91,1] = PR[GP1:90,1] + 115.580;
   1:  PR[GP1:91,2] = PR[GP1:90,2] + 90.878;
   1:L PR[91] 10mm/sec FINE;
   1:  PR[GP1:91,1] = PR[GP1:90,1] + 116.756;
   1:  PR[GP1:91,2] = PR[GP1:90,2] + 91.750;
   1:L PR[91] 10mm/sec FINE;
   1:  PR[GP1:91,1] = PR[GP1:90,1] + 117.493;
   1:  PR[GP1:91,2] = PR[GP1:90,2] + 92.439;
   1:L PR[91] 10mm/sec FINE;
   1:  PR[GP1:91,1] = PR[GP1:90,1] + 118.947;
   1:  PR[GP1:91,2] = PR[GP1:90,2] + 93.922;
   1:L PR[91] 10mm/sec FINE;
   1:  PR[GP1:91,1] = PR[GP1:90,1] + 119.642;
   1:  PR[GP1:91,2] = PR[GP1:90,2] + 94.876;
   1:L PR[91] 10mm/sec FINE;
   1:  PR[GP1:91,1] = PR[GP1:90,1] + 120.783;
   1:  PR[GP1:91,2] = PR[GP1:90,2] + 96.367;
   1:L PR[91] 10mm/sec FINE;
   1:  PR[GP1:91,1] = PR[GP1:90,1] + 122.227;
   1:  PR[GP1:91,2] = PR[GP1:90,2] + 99.015;
   1:L PR[91] 10mm/sec FINE;
   1:  PR[GP1:91,1] = PR[GP1:90,1] + 123.247;
   1:  PR[GP1:91,2] = PR[GP1:90,2] + 101.831;
   1:L PR[91] 10mm/sec FINE;
   1:  PR[GP1:91,1] = PR[GP1:90,1] + 123.579;
   1:  PR[GP1:91,2] = PR[GP1:90,2] + 103.515;
   1:L PR[91] 10mm/sec FINE;
   1:  PR[GP1:91,1] = PR[GP1:90,1] + 123.805;
   1:  PR[GP1:91,2] = PR[GP1:90,2] + 104.511;
   1:L PR[91] 10mm/sec FINE;
   1:  PR[GP1:91,1] = PR[GP1:90,1] + 123.847;
   1:  PR[GP1:91,2] = PR[GP1:90,2] + 104.719;
   1:L PR[91] 10mm/sec FINE;
   1:  PR[GP1:91,1] = PR[GP1:90,1] + 123.976;
   1:  PR[GP1:91,2] = PR[GP1:90,2] + 107.579;
   1:L PR[91] 10mm/sec FINE;
   1:  PR[GP1:91,1] = PR[GP1:90,1] + 123.523;
   1:  PR[GP1:91,2] = PR[GP1:90,2] + 111.152;
   1:L PR[91] 10mm/sec FINE;
   1:  PR[GP1:91,1] = PR[GP1:90,1] + 122.373;
   1:  PR[GP1:91,2] = PR[GP1:90,2] + 114.511;
   1:L PR[91] 10mm/sec FINE;
   1:  PR[GP1:91,1] = PR[GP1:90,1] + 120.582;
   1:  PR[GP1:91,2] = PR[GP1:90,2] + 117.521;
   1:L PR[91] 10mm/sec FINE;
   1:  PR[GP1:91,1] = PR[GP1:90,1] + 118.237;
   1:  PR[GP1:91,2] = PR[GP1:90,2] + 120.084;
   1:L PR[91] 10mm/sec FINE;
   1:  PR[GP1:91,1] = PR[GP1:90,1] + 117.790;
   1:  PR[GP1:91,2] = PR[GP1:90,2] + 120.412;
   1:L PR[91] 10mm/sec FINE;
   1:  PR[GP1:91,1] = PR[GP1:90,1] + 115.433;
   1:  PR[GP1:91,2] = PR[GP1:90,2] + 122.117;
   1:L PR[91] 10mm/sec FINE;
   1:  PR[GP1:91,1] = PR[GP1:90,1] + 112.261;
   1:  PR[GP1:91,2] = PR[GP1:90,2] + 123.561;
   1:L PR[91] 10mm/sec FINE;
   1:  PR[GP1:91,1] = PR[GP1:90,1] + 108.795;
   1:  PR[GP1:91,2] = PR[GP1:90,2] + 124.383;
   1:L PR[91] 10mm/sec FINE;
   1:  PR[GP1:91,1] = PR[GP1:90,1] + 105.329;
   1:  PR[GP1:91,2] = PR[GP1:90,2] + 124.513;
   1:L PR[91] 10mm/sec FINE;
   1:  PR[GP1:91,1] = PR[GP1:90,1] + 104.105;
   1:  PR[GP1:91,2] = PR[GP1:90,2] + 124.337;
   1:L PR[91] 10mm/sec FINE;
   1:  PR[GP1:91,1] = PR[GP1:90,1] + 101.878;
   1:  PR[GP1:91,2] = PR[GP1:90,2] + 123.985;
   1:L PR[91] 10mm/sec FINE;
   1:  PR[GP1:91,1] = PR[GP1:90,1] + 98.551;
   1:  PR[GP1:91,2] = PR[GP1:90,2] + 122.813;
   1:L PR[91] 10mm/sec FINE;
   1:  PR[GP1:91,1] = PR[GP1:90,1] + 98.158;
   1:  PR[GP1:91,2] = PR[GP1:90,2] + 122.659;
   1:L PR[91] 10mm/sec FINE;
   1:  PR[GP1:91,1] = PR[GP1:90,1] + 97.600;
   1:  PR[GP1:91,2] = PR[GP1:90,2] + 122.391;
   1:L PR[91] 10mm/sec FINE;
   1:  PR[GP1:91,1] = PR[GP1:90,1] + 96.438;
   1:  PR[GP1:91,2] = PR[GP1:90,2] + 122.155;
   1:L PR[91] 10mm/sec FINE;
   1:  PR[GP1:91,1] = PR[GP1:90,1] + 95.791;
   1:  PR[GP1:91,2] = PR[GP1:90,2] + 122.284;
   1:L PR[91] 10mm/sec FINE;
   1:  PR[GP1:91,1] = PR[GP1:90,1] + 94.534;
   1:  PR[GP1:91,2] = PR[GP1:90,2] + 122.708;
   1:L PR[91] 10mm/sec FINE;
   1:  PR[GP1:91,1] = PR[GP1:90,1] + 93.787;
   1:  PR[GP1:91,2] = PR[GP1:90,2] + 122.931;
   1:L PR[91] 10mm/sec FINE;
   1:  PR[GP1:91,1] = PR[GP1:90,1] + 90.834;
   1:  PR[GP1:91,2] = PR[GP1:90,2] + 123.632;
   1:L PR[91] 10mm/sec FINE;
   1:  PR[GP1:91,1] = PR[GP1:90,1] + 90.021;
   1:  PR[GP1:91,2] = PR[GP1:90,2] + 123.769;
   1:L PR[91] 10mm/sec FINE;
   1:  PR[GP1:91,1] = PR[GP1:90,1] + 87.284;
   1:  PR[GP1:91,2] = PR[GP1:90,2] + 124.119;
   1:L PR[91] 10mm/sec FINE;
   1:  PR[GP1:91,1] = PR[GP1:90,1] + 84.719;
   1:  PR[GP1:91,2] = PR[GP1:90,2] + 124.140;
   1:L PR[91] 10mm/sec FINE;
   1:  PR[GP1:91,1] = PR[GP1:90,1] + 83.098;
   1:  PR[GP1:91,2] = PR[GP1:90,2] + 124.014;
   1:L PR[91] 10mm/sec FINE;
   1:  PR[GP1:91,1] = PR[GP1:90,1] + 81.560;
   1:  PR[GP1:91,2] = PR[GP1:90,2] + 123.840;
   1:L PR[91] 10mm/sec FINE;
   1:  PR[GP1:91,1] = PR[GP1:90,1] + 77.890;
   1:  PR[GP1:91,2] = PR[GP1:90,2] + 122.937;
   1:L PR[91] 10mm/sec FINE;
   1:  PR[GP1:91,1] = PR[GP1:90,1] + 77.732;
   1:  PR[GP1:91,2] = PR[GP1:90,2] + 122.877;
   1:L PR[91] 10mm/sec FINE;
   1:  PR[GP1:91,1] = PR[GP1:90,1] + 76.889;
   1:  PR[GP1:91,2] = PR[GP1:90,2] + 122.498;
   1:L PR[91] 10mm/sec FINE;
   1:  PR[GP1:91,1] = PR[GP1:90,1] + 74.660;
   1:  PR[GP1:91,2] = PR[GP1:90,2] + 121.436;
   1:L PR[91] 10mm/sec FINE;
   1:  PR[GP1:91,1] = PR[GP1:90,1] + 74.096;
   1:  PR[GP1:91,2] = PR[GP1:90,2] + 121.063;
   1:L PR[91] 10mm/sec FINE;
   1:  PR[GP1:91,1] = PR[GP1:90,1] + 71.892;
   1:  PR[GP1:91,2] = PR[GP1:90,2] + 119.409;
   1:L PR[91] 10mm/sec FINE;
   1:  PR[GP1:91,1] = PR[GP1:90,1] + 70.971;
   1:  PR[GP1:91,2] = PR[GP1:90,2] + 118.452;
   1:L PR[91] 10mm/sec FINE;
   1:  PR[GP1:91,1] = PR[GP1:90,1] + 69.582;
   1:  PR[GP1:91,2] = PR[GP1:90,2] + 116.841;
   1:L PR[91] 10mm/sec FINE;
   1:  PR[GP1:91,1] = PR[GP1:90,1] + 68.712;
   1:  PR[GP1:91,2] = PR[GP1:90,2] + 115.384;
   1:L PR[91] 10mm/sec FINE;
   1:  PR[GP1:91,1] = PR[GP1:90,1] + 67.864;
   1:  PR[GP1:91,2] = PR[GP1:90,2] + 113.819;
   1:L PR[91] 10mm/sec FINE;
   1:  PR[GP1:91,1] = PR[GP1:90,1] + 67.291;
   1:  PR[GP1:91,2] = PR[GP1:90,2] + 112.076;
   1:L PR[91] 10mm/sec FINE;
   1:  PR[GP1:91,1] = PR[GP1:90,1] + 66.819;
   1:  PR[GP1:91,2] = PR[GP1:90,2] + 110.494;
   1:L PR[91] 10mm/sec FINE;
   1:  PR[GP1:91,1] = PR[GP1:90,1] + 66.724;
   1:  PR[GP1:91,2] = PR[GP1:90,2] + 108.711;
   1:L PR[91] 10mm/sec FINE;
   1:  PR[GP1:91,1] = PR[GP1:90,1] + 66.582;
   1:  PR[GP1:91,2] = PR[GP1:90,2] + 107.411;
   1:L PR[91] 10mm/sec FINE;
   1:  PR[GP1:91,1] = PR[GP1:90,1] + 66.570;
   1:  PR[GP1:91,2] = PR[GP1:90,2] + 106.986;
   1:L PR[91] 10mm/sec FINE;
   1:  PR[GP1:91,1] = PR[GP1:90,1] + 66.945;
   1:  PR[GP1:91,2] = PR[GP1:90,2] + 105.430;
   1:L PR[91] 10mm/sec FINE;
   1:  PR[GP1:91,1] = PR[GP1:90,1] + 67.342;
   1:  PR[GP1:91,2] = PR[GP1:90,2] + 103.344;
   1:L PR[91] 10mm/sec FINE;
   1:  PR[GP1:91,1] = PR[GP1:90,1] + 68.685;
   1:  PR[GP1:91,2] = PR[GP1:90,2] + 99.961;
   1:L PR[91] 10mm/sec FINE;
   1:  PR[GP1:91,1] = PR[GP1:90,1] + 70.225;
   1:  PR[GP1:91,2] = PR[GP1:90,2] + 97.666;
   1:L PR[91] 10mm/sec FINE;
   1:  PR[GP1:91,1] = PR[GP1:90,1] + 70.753;
   1:  PR[GP1:91,2] = PR[GP1:90,2] + 96.930;
   1:L PR[91] 10mm/sec FINE;
   1:  PR[GP1:91,1] = PR[GP1:90,1] + 70.883;
   1:  PR[GP1:91,2] = PR[GP1:90,2] + 96.782;
   1:L PR[91] 10mm/sec FINE;
   1:  PR[GP1:91,1] = PR[GP1:90,1] + 73.192;
   1:  PR[GP1:91,2] = PR[GP1:90,2] + 94.585;
   1:L PR[91] 10mm/sec FINE;
   1:  PR[GP1:91,1] = PR[GP1:90,1] + 74.881;
   1:  PR[GP1:91,2] = PR[GP1:90,2] + 93.567;
   1:  PR[GP1:91,3] = PR[GP1:90,3] + 36.900;
   1:L PR[91] 10mm/sec FINE;
   1:  PR[GP1:91,1] = PR[GP1:90,1] + 77.975;
   1:  PR[GP1:91,2] = PR[GP1:90,2] + 91.540;
   1:L PR[91] 10mm/sec FINE;
   1:  PR[GP1:91,1] = PR[GP1:90,1] + 80.801;
   1:  PR[GP1:91,2] = PR[GP1:90,2] + 90.167;
   1:L PR[91] 10mm/sec FINE;
   1:  PR[GP1:91,1] = PR[GP1:90,1] + 81.670;
   1:  PR[GP1:91,2] = PR[GP1:90,2] + 89.786;
   1:L PR[91] 10mm/sec FINE;
   1:  PR[GP1:91,1] = PR[GP1:90,1] + 84.243;
   1:  PR[GP1:91,2] = PR[GP1:90,2] + 88.892;
   1:L PR[91] 10mm/sec FINE;
   1:  PR[GP1:91,1] = PR[GP1:90,1] + 86.637;
   1:  PR[GP1:91,2] = PR[GP1:90,2] + 88.319;
   1:L PR[91] 10mm/sec FINE;
   1:  PR[GP1:91,1] = PR[GP1:90,1] + 88.545;
   1:  PR[GP1:91,2] = PR[GP1:90,2] + 87.911;
   1:L PR[91] 10mm/sec FINE;
   1:  PR[GP1:91,1] = PR[GP1:90,1] + 89.822;
   1:  PR[GP1:91,2] = PR[GP1:90,2] + 87.798;
   1:L PR[91] 10mm/sec FINE;
   1:  PR[GP1:91,1] = PR[GP1:90,1] + 93.804;
   1:  PR[GP1:91,2] = PR[GP1:90,2] + 87.589;
   1:L PR[91] 10mm/sec FINE;
   1:  PR[GP1:91,1] = PR[GP1:90,1] + 94.261;
   1:  PR[GP1:91,2] = PR[GP1:90,2] + 87.606;
   1:L PR[91] 10mm/sec FINE;
   1:  PR[GP1:91,1] = PR[GP1:90,1] + 96.741;
   1:  PR[GP1:91,2] = PR[GP1:90,2] + 87.961;
   1:L PR[91] 10mm/sec FINE;
   1:  PR[GP1:91,1] = PR[GP1:90,1] + 98.861;
   1:  PR[GP1:91,2] = PR[GP1:90,2] + 88.154;
   1:L PR[91] 10mm/sec FINE;
   1:  PR[GP1:91,1] = PR[GP1:90,1] + 99.964;
   1:  PR[GP1:91,2] = PR[GP1:90,2] + 88.083;
   1:L PR[91] 10mm/sec FINE;
   1:  PR[GP1:91,1] = PR[GP1:90,1] + 102.646;
   1:  PR[GP1:91,2] = PR[GP1:90,2] + 87.457;
   1:L PR[91] 10mm/sec FINE;
   1:  PR[GP1:91,1] = PR[GP1:90,1] + 102.888;
   1:  PR[GP1:91,2] = PR[GP1:90,2] + 87.420;
   1:L PR[91] 10mm/sec FINE;
   1:  PR[GP1:91,1] = PR[GP1:90,1] + 105.492;
   1:  PR[GP1:91,2] = PR[GP1:90,2] + 87.254;
   1:L PR[91] 10mm/sec FINE;
   1:  PR[GP1:91,1] = PR[GP1:90,1] + 105.799;
   1:  PR[GP1:91,2] = PR[GP1:90,2] + 87.256;
   1:L PR[91] 10mm/sec FINE;
   1:  PR[GP1:91,1] = PR[GP1:90,1] + 108.370;
   1:  PR[GP1:91,2] = PR[GP1:90,2] + 87.524;
   1:L PR[91] 10mm/sec FINE;
   1:  PR[GP1:91,1] = PR[GP1:90,1] + 108.651;
   1:  PR[GP1:91,2] = PR[GP1:90,2] + 87.571;
   1:L PR[91] 10mm/sec FINE;
   1:  PR[GP1:91,1] = PR[GP1:90,1] + 111.233;
   1:  PR[GP1:91,2] = PR[GP1:90,2] + 88.295;
   1:L PR[91] 10mm/sec FINE;
   1:  PR[GP1:91,1] = PR[GP1:90,1] + 111.383;
   1:  PR[GP1:91,2] = PR[GP1:90,2] + 88.346;
   1:L PR[91] 10mm/sec FINE;
   1:  PR[GP1:91,1] = PR[GP1:90,1] + 113.918;
   1:  PR[GP1:91,2] = PR[GP1:90,2] + 89.533;
   1:L PR[91] 10mm/sec FINE;
   1:  PR[GP1:91,1] = PR[GP1:90,1] + 116.130;
   1:  PR[GP1:91,2] = PR[GP1:90,2] + 91.007;
   1:L PR[91] 10mm/sec FINE;
   1:  PR[GP1:91,1] = PR[GP1:90,1] + 116.519;
   1:  PR[GP1:91,2] = PR[GP1:90,2] + 91.295;
   1:L PR[91] 10mm/sec FINE;
   1:  PR[GP1:91,1] = PR[GP1:90,1] + 118.018;
   1:  PR[GP1:91,2] = PR[GP1:90,2] + 92.695;
   1:L PR[91] 10mm/sec FINE;
   1:  PR[GP1:91,1] = PR[GP1:90,1] + 118.747;
   1:  PR[GP1:91,2] = PR[GP1:90,2] + 93.439;
   1:L PR[91] 10mm/sec FINE;
   1:  PR[GP1:91,1] = PR[GP1:90,1] + 119.594;
   1:  PR[GP1:91,2] = PR[GP1:90,2] + 94.530;
   1:L PR[91] 10mm/sec FINE;
   1:  PR[GP1:91,1] = PR[GP1:90,1] + 120.596;
   1:  PR[GP1:91,2] = PR[GP1:90,2] + 95.936;
   1:L PR[91] 10mm/sec FINE;
   1:  PR[GP1:91,1] = PR[GP1:90,1] + 120.887;
   1:  PR[GP1:91,2] = PR[GP1:90,2] + 96.464;
   1:L PR[91] 10mm/sec FINE;
   1:  PR[GP1:91,1] = PR[GP1:90,1] + 121.660;
   1:  PR[GP1:91,2] = PR[GP1:90,2] + 97.999;
   1:L PR[91] 10mm/sec FINE;
   1:  PR[GP1:91,1] = PR[GP1:90,1] + 122.027;
   1:  PR[GP1:91,2] = PR[GP1:90,2] + 98.667;
   1:L PR[91] 10mm/sec FINE;
   1:  PR[GP1:91,1] = PR[GP1:90,1] + 123.067;
   1:  PR[GP1:91,2] = PR[GP1:90,2] + 101.481;
   1:L PR[91] 10mm/sec FINE;
   1:  PR[GP1:91,1] = PR[GP1:90,1] + 123.655;
   1:  PR[GP1:91,2] = PR[GP1:90,2] + 104.385;
   1:L PR[91] 10mm/sec FINE;
   1:  PR[GP1:91,1] = PR[GP1:90,1] + 123.749;
   1:  PR[GP1:91,2] = PR[GP1:90,2] + 107.316;
   1:L PR[91] 10mm/sec FINE;
   1:  PR[GP1:91,1] = PR[GP1:90,1] + 123.531;
   1:  PR[GP1:91,2] = PR[GP1:90,2] + 109.195;
   1:L PR[91] 10mm/sec FINE;
   1:  PR[GP1:91,1] = PR[GP1:90,1] + 123.310;
   1:  PR[GP1:91,2] = PR[GP1:90,2] + 110.901;
   1:L PR[91] 10mm/sec FINE;
   1:  PR[GP1:91,1] = PR[GP1:90,1] + 122.171;
   1:  PR[GP1:91,2] = PR[GP1:90,2] + 114.273;
   1:L PR[91] 10mm/sec FINE;
   1:  PR[GP1:91,1] = PR[GP1:90,1] + 120.382;
   1:  PR[GP1:91,2] = PR[GP1:90,2] + 117.299;
   1:L PR[91] 10mm/sec FINE;
   1:  PR[GP1:91,1] = PR[GP1:90,1] + 118.031;
   1:  PR[GP1:91,2] = PR[GP1:90,2] + 119.877;
   1:L PR[91] 10mm/sec FINE;
   1:  PR[GP1:91,1] = PR[GP1:90,1] + 116.657;
   1:  PR[GP1:91,2] = PR[GP1:90,2] + 120.884;
   1:L PR[91] 10mm/sec FINE;
   1:  PR[GP1:91,1] = PR[GP1:90,1] + 115.218;
   1:  PR[GP1:91,2] = PR[GP1:90,2] + 121.925;
   1:L PR[91] 10mm/sec FINE;
   1:  PR[GP1:91,1] = PR[GP1:90,1] + 112.031;
   1:  PR[GP1:91,2] = PR[GP1:90,2] + 123.382;
   1:L PR[91] 10mm/sec FINE;
   1:  PR[GP1:91,1] = PR[GP1:90,1] + 108.648;
   1:  PR[GP1:91,2] = PR[GP1:90,2] + 124.189;
   1:L PR[91] 10mm/sec FINE;
   1:  PR[GP1:91,1] = PR[GP1:90,1] + 105.107;
   1:  PR[GP1:91,2] = PR[GP1:90,2] + 124.345;
   1:L PR[91] 10mm/sec FINE;
   1:  PR[GP1:91,1] = PR[GP1:90,1] + 101.722;
   1:  PR[GP1:91,2] = PR[GP1:90,2] + 123.810;
   1:L PR[91] 10mm/sec FINE;
   1:  PR[GP1:91,1] = PR[GP1:90,1] + 98.396;
   1:  PR[GP1:91,2] = PR[GP1:90,2] + 122.646;
   1:L PR[91] 10mm/sec FINE;
   1:  PR[GP1:91,1] = PR[GP1:90,1] + 97.775;
   1:  PR[GP1:91,2] = PR[GP1:90,2] + 122.397;
   1:L PR[91] 10mm/sec FINE;
   1:  PR[GP1:91,1] = PR[GP1:90,1] + 96.621;
   1:  PR[GP1:91,2] = PR[GP1:90,2] + 122.164;
   1:L PR[91] 10mm/sec FINE;
   1:  PR[GP1:91,1] = PR[GP1:90,1] + 96.039;
   1:  PR[GP1:91,2] = PR[GP1:90,2] + 122.292;
   1:L PR[91] 10mm/sec FINE;
   1:  PR[GP1:91,1] = PR[GP1:90,1] + 95.648;
   1:  PR[GP1:91,2] = PR[GP1:90,2] + 122.423;
   1:L PR[91] 10mm/sec FINE;
   1:  PR[GP1:91,1] = PR[GP1:90,1] + 94.661;
   1:  PR[GP1:91,2] = PR[GP1:90,2] + 122.719;
   1:L PR[91] 10mm/sec FINE;
   1:  PR[GP1:91,1] = PR[GP1:90,1] + 94.205;
   1:  PR[GP1:91,2] = PR[GP1:90,2] + 122.836;
   1:L PR[91] 10mm/sec FINE;
   1:  PR[GP1:91,1] = PR[GP1:90,1] + 91.910;
   1:  PR[GP1:91,2] = PR[GP1:90,2] + 123.372;
   1:L PR[91] 10mm/sec FINE;
   1:  PR[GP1:91,1] = PR[GP1:90,1] + 90.561;
   1:  PR[GP1:91,2] = PR[GP1:90,2] + 123.599;
   1:L PR[91] 10mm/sec FINE;
   1:  PR[GP1:91,1] = PR[GP1:90,1] + 88.098;
   1:  PR[GP1:91,2] = PR[GP1:90,2] + 123.915;
   1:L PR[91] 10mm/sec FINE;
   1:  PR[GP1:91,1] = PR[GP1:90,1] + 85.129;
   1:  PR[GP1:91,2] = PR[GP1:90,2] + 123.960;
   1:L PR[91] 10mm/sec FINE;
   1:  PR[GP1:91,1] = PR[GP1:90,1] + 84.505;
   1:  PR[GP1:91,2] = PR[GP1:90,2] + 123.912;
   1:L PR[91] 10mm/sec FINE;
   1:  PR[GP1:91,1] = PR[GP1:90,1] + 82.183;
   1:  PR[GP1:91,2] = PR[GP1:90,2] + 123.649;
   1:L PR[91] 10mm/sec FINE;
   1:  PR[GP1:91,1] = PR[GP1:90,1] + 78.729;
   1:  PR[GP1:91,2] = PR[GP1:90,2] + 122.798;
   1:L PR[91] 10mm/sec FINE;
   1:  PR[GP1:91,1] = PR[GP1:90,1] + 78.109;
   1:  PR[GP1:91,2] = PR[GP1:90,2] + 122.561;
   1:L PR[91] 10mm/sec FINE;
   1:  PR[GP1:91,1] = PR[GP1:90,1] + 75.047;
   1:  PR[GP1:91,2] = PR[GP1:90,2] + 121.183;
   1:L PR[91] 10mm/sec FINE;
   1:  PR[GP1:91,1] = PR[GP1:90,1] + 72.331;
   1:  PR[GP1:91,2] = PR[GP1:90,2] + 119.147;
   1:L PR[91] 10mm/sec FINE;
   1:  PR[GP1:91,1] = PR[GP1:90,1] + 71.861;
   1:  PR[GP1:91,2] = PR[GP1:90,2] + 118.658;
   1:L PR[91] 10mm/sec FINE;
   1:  PR[GP1:91,1] = PR[GP1:90,1] + 70.072;
   1:  PR[GP1:91,2] = PR[GP1:90,2] + 116.583;
   1:L PR[91] 10mm/sec FINE;
   1:  PR[GP1:91,1] = PR[GP1:90,1] + 69.515;
   1:  PR[GP1:91,2] = PR[GP1:90,2] + 115.650;
   1:L PR[91] 10mm/sec FINE;
   1:  PR[GP1:91,1] = PR[GP1:90,1] + 68.391;
   1:  PR[GP1:91,2] = PR[GP1:90,2] + 113.578;
   1:L PR[91] 10mm/sec FINE;
   1:  PR[GP1:91,1] = PR[GP1:90,1] + 67.999;
   1:  PR[GP1:91,2] = PR[GP1:90,2] + 112.385;
   1:L PR[91] 10mm/sec FINE;
   1:  PR[GP1:91,1] = PR[GP1:90,1] + 67.370;
   1:  PR[GP1:91,2] = PR[GP1:90,2] + 110.280;
   1:L PR[91] 10mm/sec FINE;
   1:  PR[GP1:91,1] = PR[GP1:90,1] + 67.305;
   1:  PR[GP1:91,2] = PR[GP1:90,2] + 109.051;
   1:L PR[91] 10mm/sec FINE;
   1:  PR[GP1:91,1] = PR[GP1:90,1] + 67.206;
   1:  PR[GP1:91,2] = PR[GP1:90,2] + 108.151;
   1:L PR[91] 10mm/sec FINE;
   1:  PR[GP1:91,1] = PR[GP1:90,1] + 67.169;
   1:  PR[GP1:91,2] = PR[GP1:90,2] + 106.792;
   1:L PR[91] 10mm/sec FINE;
   1:  PR[GP1:91,1] = PR[GP1:90,1] + 67.411;
   1:  PR[GP1:91,2] = PR[GP1:90,2] + 105.790;
   1:L PR[91] 10mm/sec FINE;
   1:  PR[GP1:91,1] = PR[GP1:90,1] + 67.906;
   1:  PR[GP1:91,2] = PR[GP1:90,2] + 103.188;
   1:L PR[91] 10mm/sec FINE;
   1:  PR[GP1:91,1] = PR[GP1:90,1] + 69.228;
   1:  PR[GP1:91,2] = PR[GP1:90,2] + 99.836;
   1:L PR[91] 10mm/sec FINE;
   1:  PR[GP1:91,1] = PR[GP1:90,1] + 71.291;
   1:  PR[GP1:91,2] = PR[GP1:90,2] + 96.958;
   1:L PR[91] 10mm/sec FINE;
   1:  PR[GP1:91,1] = PR[GP1:90,1] + 71.814;
   1:  PR[GP1:91,2] = PR[GP1:90,2] + 96.362;
   1:L PR[91] 10mm/sec FINE;
   1:  PR[GP1:91,1] = PR[GP1:90,1] + 73.597;
   1:  PR[GP1:91,2] = PR[GP1:90,2] + 94.666;
   1:L PR[91] 10mm/sec FINE;
   1:  PR[GP1:91,1] = PR[GP1:90,1] + 75.716;
   1:  PR[GP1:91,2] = PR[GP1:90,2] + 93.278;
   1:  PR[GP1:91,3] = PR[GP1:90,3] + 37.900;
   1:L PR[91] 10mm/sec FINE;
   1:  PR[GP1:91,1] = PR[GP1:90,1] + 76.166;
   1:  PR[GP1:91,2] = PR[GP1:90,2] + 92.979;
   1:L PR[91] 10mm/sec FINE;
   1:  PR[GP1:91,1] = PR[GP1:90,1] + 78.792;
   1:  PR[GP1:91,2] = PR[GP1:90,2] + 91.271;
   1:L PR[91] 10mm/sec FINE;
   1:  PR[GP1:91,1] = PR[GP1:90,1] + 81.331;
   1:  PR[GP1:91,2] = PR[GP1:90,2] + 90.036;
   1:L PR[91] 10mm/sec FINE;
   1:  PR[GP1:91,1] = PR[GP1:90,1] + 82.714;
   1:  PR[GP1:91,2] = PR[GP1:90,2] + 89.429;
   1:L PR[91] 10mm/sec FINE;
   1:  PR[GP1:91,1] = PR[GP1:90,1] + 84.900;
   1:  PR[GP1:91,2] = PR[GP1:90,2] + 88.670;
   1:L PR[91] 10mm/sec FINE;
   1:  PR[GP1:91,1] = PR[GP1:90,1] + 87.969;
   1:  PR[GP1:91,2] = PR[GP1:90,2] + 87.936;
   1:L PR[91] 10mm/sec FINE;
   1:  PR[GP1:91,1] = PR[GP1:90,1] + 89.382;
   1:  PR[GP1:91,2] = PR[GP1:90,2] + 87.634;
   1:L PR[91] 10mm/sec FINE;
   1:  PR[GP1:91,1] = PR[GP1:90,1] + 90.325;
   1:  PR[GP1:91,2] = PR[GP1:90,2] + 87.551;
   1:L PR[91] 10mm/sec FINE;
   1:  PR[GP1:91,1] = PR[GP1:90,1] + 94.852;
   1:  PR[GP1:91,2] = PR[GP1:90,2] + 87.313;
   1:L PR[91] 10mm/sec FINE;
   1:  PR[GP1:91,1] = PR[GP1:90,1] + 95.353;
   1:  PR[GP1:91,2] = PR[GP1:90,2] + 87.376;
   1:L PR[91] 10mm/sec FINE;
   1:  PR[GP1:91,1] = PR[GP1:90,1] + 99.305;
   1:  PR[GP1:91,2] = PR[GP1:90,2] + 87.739;
   1:L PR[91] 10mm/sec FINE;
   1:  PR[GP1:91,1] = PR[GP1:90,1] + 100.335;
   1:  PR[GP1:91,2] = PR[GP1:90,2] + 87.673;
   1:L PR[91] 10mm/sec FINE;
   1:  PR[GP1:91,1] = PR[GP1:90,1] + 102.398;
   1:  PR[GP1:91,2] = PR[GP1:90,2] + 87.203;
   1:L PR[91] 10mm/sec FINE;
   1:  PR[GP1:91,1] = PR[GP1:90,1] + 103.288;
   1:  PR[GP1:91,2] = PR[GP1:90,2] + 87.070;
   1:L PR[91] 10mm/sec FINE;
   1:  PR[GP1:91,1] = PR[GP1:90,1] + 105.177;
   1:  PR[GP1:91,2] = PR[GP1:90,2] + 86.949;
   1:L PR[91] 10mm/sec FINE;
   1:  PR[GP1:91,1] = PR[GP1:90,1] + 106.185;
   1:  PR[GP1:91,2] = PR[GP1:90,2] + 86.957;
   1:L PR[91] 10mm/sec FINE;
   1:  PR[GP1:91,1] = PR[GP1:90,1] + 107.981;
   1:  PR[GP1:91,2] = PR[GP1:90,2] + 87.144;
   1:L PR[91] 10mm/sec FINE;
   1:  PR[GP1:91,1] = PR[GP1:90,1] + 109.016;
   1:  PR[GP1:91,2] = PR[GP1:90,2] + 87.317;
   1:L PR[91] 10mm/sec FINE;
   1:  PR[GP1:91,1] = PR[GP1:90,1] + 110.768;
   1:  PR[GP1:91,2] = PR[GP1:90,2] + 87.809;
   1:L PR[91] 10mm/sec FINE;
   1:  PR[GP1:91,1] = PR[GP1:90,1] + 111.715;
   1:  PR[GP1:91,2] = PR[GP1:90,2] + 88.127;
   1:L PR[91] 10mm/sec FINE;
   1:  PR[GP1:91,1] = PR[GP1:90,1] + 113.496;
   1:  PR[GP1:91,2] = PR[GP1:90,2] + 88.970;
   1:L PR[91] 10mm/sec FINE;
   1:  PR[GP1:91,1] = PR[GP1:90,1] + 114.231;
   1:  PR[GP1:91,2] = PR[GP1:90,2] + 89.354;
   1:L PR[91] 10mm/sec FINE;
   1:  PR[GP1:91,1] = PR[GP1:90,1] + 116.117;
   1:  PR[GP1:91,2] = PR[GP1:90,2] + 90.671;
   1:L PR[91] 10mm/sec FINE;
   1:  PR[GP1:91,1] = PR[GP1:90,1] + 116.518;
   1:  PR[GP1:91,2] = PR[GP1:90,2] + 90.970;
   1:L PR[91] 10mm/sec FINE;
   1:  PR[GP1:91,1] = PR[GP1:90,1] + 118.547;
   1:  PR[GP1:91,2] = PR[GP1:90,2] + 92.956;
   1:L PR[91] 10mm/sec FINE;
   1:  PR[GP1:91,1] = PR[GP1:90,1] + 120.062;
   1:  PR[GP1:91,2] = PR[GP1:90,2] + 94.909;
   1:L PR[91] 10mm/sec FINE;
   1:  PR[GP1:91,1] = PR[GP1:90,1] + 120.436;
   1:  PR[GP1:91,2] = PR[GP1:90,2] + 95.433;
   1:L PR[91] 10mm/sec FINE;
   1:  PR[GP1:91,1] = PR[GP1:90,1] + 121.272;
   1:  PR[GP1:91,2] = PR[GP1:90,2] + 96.950;
   1:L PR[91] 10mm/sec FINE;
   1:  PR[GP1:91,1] = PR[GP1:90,1] + 121.897;
   1:  PR[GP1:91,2] = PR[GP1:90,2] + 98.189;
   1:L PR[91] 10mm/sec FINE;
   1:  PR[GP1:91,1] = PR[GP1:90,1] + 122.213;
   1:  PR[GP1:91,2] = PR[GP1:90,2] + 99.047;
   1:L PR[91] 10mm/sec FINE;
   1:  PR[GP1:91,1] = PR[GP1:90,1] + 122.897;
   1:  PR[GP1:91,2] = PR[GP1:90,2] + 101.113;
   1:L PR[91] 10mm/sec FINE;
   1:  PR[GP1:91,1] = PR[GP1:90,1] + 123.495;
   1:  PR[GP1:91,2] = PR[GP1:90,2] + 104.034;
   1:L PR[91] 10mm/sec FINE;
   1:  PR[GP1:91,1] = PR[GP1:90,1] + 123.537;
   1:  PR[GP1:91,2] = PR[GP1:90,2] + 105.649;
   1:L PR[91] 10mm/sec FINE;
   1:  PR[GP1:91,1] = PR[GP1:90,1] + 123.591;
   1:  PR[GP1:91,2] = PR[GP1:90,2] + 106.987;
   1:L PR[91] 10mm/sec FINE;
   1:  PR[GP1:91,1] = PR[GP1:90,1] + 123.272;
   1:  PR[GP1:91,2] = PR[GP1:90,2] + 109.241;
   1:L PR[91] 10mm/sec FINE;
   1:  PR[GP1:91,1] = PR[GP1:90,1] + 123.097;
   1:  PR[GP1:91,2] = PR[GP1:90,2] + 110.651;
   1:L PR[91] 10mm/sec FINE;
   1:  PR[GP1:91,1] = PR[GP1:90,1] + 121.969;
   1:  PR[GP1:91,2] = PR[GP1:90,2] + 114.035;
   1:L PR[91] 10mm/sec FINE;
   1:  PR[GP1:91,1] = PR[GP1:90,1] + 120.181;
   1:  PR[GP1:91,2] = PR[GP1:90,2] + 117.076;
   1:L PR[91] 10mm/sec FINE;
   1:  PR[GP1:91,1] = PR[GP1:90,1] + 117.825;
   1:  PR[GP1:91,2] = PR[GP1:90,2] + 119.670;
   1:L PR[91] 10mm/sec FINE;
   1:  PR[GP1:91,1] = PR[GP1:90,1] + 115.003;
   1:  PR[GP1:91,2] = PR[GP1:90,2] + 121.732;
   1:L PR[91] 10mm/sec FINE;
   1:  PR[GP1:91,1] = PR[GP1:90,1] + 111.833;
   1:  PR[GP1:91,2] = PR[GP1:90,2] + 123.194;
   1:L PR[91] 10mm/sec FINE;
   1:  PR[GP1:91,1] = PR[GP1:90,1] + 108.511;
   1:  PR[GP1:91,2] = PR[GP1:90,2] + 123.992;
   1:L PR[91] 10mm/sec FINE;
   1:  PR[GP1:91,1] = PR[GP1:90,1] + 105.015;
   1:  PR[GP1:91,2] = PR[GP1:90,2] + 124.148;
   1:L PR[91] 10mm/sec FINE;
   1:  PR[GP1:91,1] = PR[GP1:90,1] + 103.348;
   1:  PR[GP1:91,2] = PR[GP1:90,2] + 123.917;
   1:L PR[91] 10mm/sec FINE;
   1:  PR[GP1:91,1] = PR[GP1:90,1] + 101.567;
   1:  PR[GP1:91,2] = PR[GP1:90,2] + 123.635;
   1:L PR[91] 10mm/sec FINE;
   1:  PR[GP1:91,1] = PR[GP1:90,1] + 97.965;
   1:  PR[GP1:91,2] = PR[GP1:90,2] + 122.371;
   1:L PR[91] 10mm/sec FINE;
   1:  PR[GP1:91,1] = PR[GP1:90,1] + 96.807;
   1:  PR[GP1:91,2] = PR[GP1:90,2] + 122.169;
   1:L PR[91] 10mm/sec FINE;
   1:  PR[GP1:91,1] = PR[GP1:90,1] + 96.303;
   1:  PR[GP1:91,2] = PR[GP1:90,2] + 122.276;
   1:L PR[91] 10mm/sec FINE;
   1:  PR[GP1:91,1] = PR[GP1:90,1] + 95.537;
   1:  PR[GP1:91,2] = PR[GP1:90,2] + 122.505;
   1:L PR[91] 10mm/sec FINE;
   1:  PR[GP1:91,1] = PR[GP1:90,1] + 94.970;
   1:  PR[GP1:91,2] = PR[GP1:90,2] + 122.651;
   1:L PR[91] 10mm/sec FINE;
   1:  PR[GP1:91,1] = PR[GP1:90,1] + 92.986;
   1:  PR[GP1:91,2] = PR[GP1:90,2] + 123.112;
   1:L PR[91] 10mm/sec FINE;
   1:  PR[GP1:91,1] = PR[GP1:90,1] + 91.101;
   1:  PR[GP1:91,2] = PR[GP1:90,2] + 123.429;
   1:L PR[91] 10mm/sec FINE;
   1:  PR[GP1:91,1] = PR[GP1:90,1] + 88.963;
   1:  PR[GP1:91,2] = PR[GP1:90,2] + 123.703;
   1:L PR[91] 10mm/sec FINE;
   1:  PR[GP1:91,1] = PR[GP1:90,1] + 85.642;
   1:  PR[GP1:91,2] = PR[GP1:90,2] + 123.767;
   1:L PR[91] 10mm/sec FINE;
   1:  PR[GP1:91,1] = PR[GP1:90,1] + 84.942;
   1:  PR[GP1:91,2] = PR[GP1:90,2] + 123.700;
   1:L PR[91] 10mm/sec FINE;
   1:  PR[GP1:91,1] = PR[GP1:90,1] + 82.806;
   1:  PR[GP1:91,2] = PR[GP1:90,2] + 123.457;
   1:L PR[91] 10mm/sec FINE;
   1:  PR[GP1:91,1] = PR[GP1:90,1] + 79.567;
   1:  PR[GP1:91,2] = PR[GP1:90,2] + 122.659;
   1:L PR[91] 10mm/sec FINE;
   1:  PR[GP1:91,1] = PR[GP1:90,1] + 78.486;
   1:  PR[GP1:91,2] = PR[GP1:90,2] + 122.246;
   1:L PR[91] 10mm/sec FINE;
   1:  PR[GP1:91,1] = PR[GP1:90,1] + 76.065;
   1:  PR[GP1:91,2] = PR[GP1:90,2] + 121.157;
   1:L PR[91] 10mm/sec FINE;
   1:  PR[GP1:91,1] = PR[GP1:90,1] + 75.605;
   1:  PR[GP1:91,2] = PR[GP1:90,2] + 120.905;
   1:L PR[91] 10mm/sec FINE;
   1:  PR[GP1:91,1] = PR[GP1:90,1] + 72.772;
   1:  PR[GP1:91,2] = PR[GP1:90,2] + 118.885;
   1:L PR[91] 10mm/sec FINE;
   1:  PR[GP1:91,1] = PR[GP1:90,1] + 70.561;
   1:  PR[GP1:91,2] = PR[GP1:90,2] + 116.325;
   1:L PR[91] 10mm/sec FINE;
   1:  PR[GP1:91,1] = PR[GP1:90,1] + 70.317;
   1:  PR[GP1:91,2] = PR[GP1:90,2] + 115.916;
   1:L PR[91] 10mm/sec FINE;
   1:  PR[GP1:91,1] = PR[GP1:90,1] + 68.919;
   1:  PR[GP1:91,2] = PR[GP1:90,2] + 113.338;
   1:L PR[91] 10mm/sec FINE;
   1:  PR[GP1:91,1] = PR[GP1:90,1] + 68.707;
   1:  PR[GP1:91,2] = PR[GP1:90,2] + 112.694;
   1:L PR[91] 10mm/sec FINE;
   1:  PR[GP1:91,1] = PR[GP1:90,1] + 67.922;
   1:  PR[GP1:91,2] = PR[GP1:90,2] + 110.066;
   1:L PR[91] 10mm/sec FINE;
   1:  PR[GP1:91,1] = PR[GP1:90,1] + 67.886;
   1:  PR[GP1:91,2] = PR[GP1:90,2] + 109.390;
   1:L PR[91] 10mm/sec FINE;
   1:  PR[GP1:91,1] = PR[GP1:90,1] + 67.831;
   1:  PR[GP1:91,2] = PR[GP1:90,2] + 108.891;
   1:L PR[91] 10mm/sec FINE;
   1:  PR[GP1:91,1] = PR[GP1:90,1] + 67.769;
   1:  PR[GP1:91,2] = PR[GP1:90,2] + 106.597;
   1:L PR[91] 10mm/sec FINE;
   1:  PR[GP1:91,1] = PR[GP1:90,1] + 67.876;
   1:  PR[GP1:91,2] = PR[GP1:90,2] + 106.150;
   1:L PR[91] 10mm/sec FINE;
   1:  PR[GP1:91,1] = PR[GP1:90,1] + 68.470;
   1:  PR[GP1:91,2] = PR[GP1:90,2] + 103.035;
   1:L PR[91] 10mm/sec FINE;
   1:  PR[GP1:91,1] = PR[GP1:90,1] + 69.880;
   1:  PR[GP1:91,2] = PR[GP1:90,2] + 99.759;
   1:L PR[91] 10mm/sec FINE;
   1:  PR[GP1:91,1] = PR[GP1:90,1] + 70.175;
   1:  PR[GP1:91,2] = PR[GP1:90,2] + 99.289;
   1:L PR[91] 10mm/sec FINE;
   1:  PR[GP1:91,1] = PR[GP1:90,1] + 71.828;
   1:  PR[GP1:91,2] = PR[GP1:90,2] + 96.987;
   1:L PR[91] 10mm/sec FINE;
   1:  PR[GP1:91,1] = PR[GP1:90,1] + 72.745;
   1:  PR[GP1:91,2] = PR[GP1:90,2] + 95.942;
   1:L PR[91] 10mm/sec FINE;
   1:  PR[GP1:91,1] = PR[GP1:90,1] + 74.001;
   1:  PR[GP1:91,2] = PR[GP1:90,2] + 94.747;
   1:L PR[91] 10mm/sec FINE;
   1:  PR[GP1:91,1] = PR[GP1:90,1] + 76.525;
   1:  PR[GP1:91,2] = PR[GP1:90,2] + 93.012;
   1:  PR[GP1:91,3] = PR[GP1:90,3] + 38.900;
   1:L PR[91] 10mm/sec FINE;
   1:  PR[GP1:91,1] = PR[GP1:90,1] + 76.616;
   1:  PR[GP1:91,2] = PR[GP1:90,2] + 92.950;
   1:L PR[91] 10mm/sec FINE;
   1:  PR[GP1:91,1] = PR[GP1:90,1] + 79.622;
   1:  PR[GP1:91,2] = PR[GP1:90,2] + 90.994;
   1:L PR[91] 10mm/sec FINE;
   1:  PR[GP1:91,1] = PR[GP1:90,1] + 81.861;
   1:  PR[GP1:91,2] = PR[GP1:90,2] + 89.906;
   1:L PR[91] 10mm/sec FINE;
   1:  PR[GP1:91,1] = PR[GP1:90,1] + 83.758;
   1:  PR[GP1:91,2] = PR[GP1:90,2] + 89.073;
   1:L PR[91] 10mm/sec FINE;
   1:  PR[GP1:91,1] = PR[GP1:90,1] + 85.558;
   1:  PR[GP1:91,2] = PR[GP1:90,2] + 88.448;
   1:L PR[91] 10mm/sec FINE;
   1:  PR[GP1:91,1] = PR[GP1:90,1] + 89.301;
   1:  PR[GP1:91,2] = PR[GP1:90,2] + 87.553;
   1:L PR[91] 10mm/sec FINE;
   1:  PR[GP1:91,1] = PR[GP1:90,1] + 90.218;
   1:  PR[GP1:91,2] = PR[GP1:90,2] + 87.357;
   1:L PR[91] 10mm/sec FINE;
   1:  PR[GP1:91,1] = PR[GP1:90,1] + 90.828;
   1:  PR[GP1:91,2] = PR[GP1:90,2] + 87.303;
   1:L PR[91] 10mm/sec FINE;
   1:  PR[GP1:91,1] = PR[GP1:90,1] + 94.115;
   1:  PR[GP1:91,2] = PR[GP1:90,2] + 87.130;
   1:L PR[91] 10mm/sec FINE;
   1:  PR[GP1:91,1] = PR[GP1:90,1] + 95.487;
   1:  PR[GP1:91,2] = PR[GP1:90,2] + 86.982;
   1:L PR[91] 10mm/sec FINE;
   1:  PR[GP1:91,1] = PR[GP1:90,1] + 95.896;
   1:  PR[GP1:91,2] = PR[GP1:90,2] + 86.965;
   1:L PR[91] 10mm/sec FINE;
   1:  PR[GP1:91,1] = PR[GP1:90,1] + 99.766;
   1:  PR[GP1:91,2] = PR[GP1:90,2] + 87.328;
   1:L PR[91] 10mm/sec FINE;
   1:  PR[GP1:91,1] = PR[GP1:90,1] + 100.725;
   1:  PR[GP1:91,2] = PR[GP1:90,2] + 87.267;
   1:L PR[91] 10mm/sec FINE;
   1:  PR[GP1:91,1] = PR[GP1:90,1] + 102.151;
   1:  PR[GP1:91,2] = PR[GP1:90,2] + 86.950;
   1:L PR[91] 10mm/sec FINE;
   1:  PR[GP1:91,1] = PR[GP1:90,1] + 103.687;
   1:  PR[GP1:91,2] = PR[GP1:90,2] + 86.719;
   1:L PR[91] 10mm/sec FINE;
   1:  PR[GP1:91,1] = PR[GP1:90,1] + 104.861;
   1:  PR[GP1:91,2] = PR[GP1:90,2] + 86.644;
   1:L PR[91] 10mm/sec FINE;
   1:  PR[GP1:91,1] = PR[GP1:90,1] + 106.572;
   1:  PR[GP1:91,2] = PR[GP1:90,2] + 86.657;
   1:L PR[91] 10mm/sec FINE;
   1:  PR[GP1:91,1] = PR[GP1:90,1] + 107.591;
   1:  PR[GP1:91,2] = PR[GP1:90,2] + 86.764;
   1:L PR[91] 10mm/sec FINE;
   1:  PR[GP1:91,1] = PR[GP1:90,1] + 109.380;
   1:  PR[GP1:91,2] = PR[GP1:90,2] + 87.063;
   1:L PR[91] 10mm/sec FINE;
   1:  PR[GP1:91,1] = PR[GP1:90,1] + 110.303;
   1:  PR[GP1:91,2] = PR[GP1:90,2] + 87.322;
   1:L PR[91] 10mm/sec FINE;
   1:  PR[GP1:91,1] = PR[GP1:90,1] + 112.047;
   1:  PR[GP1:91,2] = PR[GP1:90,2] + 87.909;
   1:L PR[91] 10mm/sec FINE;
   1:  PR[GP1:91,1] = PR[GP1:90,1] + 112.959;
   1:  PR[GP1:91,2] = PR[GP1:90,2] + 88.340;
   1:L PR[91] 10mm/sec FINE;
   1:  PR[GP1:91,1] = PR[GP1:90,1] + 114.524;
   1:  PR[GP1:91,2] = PR[GP1:90,2] + 89.160;
   1:L PR[91] 10mm/sec FINE;
   1:  PR[GP1:91,1] = PR[GP1:90,1] + 115.518;
   1:  PR[GP1:91,2] = PR[GP1:90,2] + 89.854;
   1:L PR[91] 10mm/sec FINE;
   1:  PR[GP1:91,1] = PR[GP1:90,1] + 116.766;
   1:  PR[GP1:91,2] = PR[GP1:90,2] + 90.783;
   1:L PR[91] 10mm/sec FINE;
   1:  PR[GP1:91,1] = PR[GP1:90,1] + 117.927;
   1:  PR[GP1:91,2] = PR[GP1:90,2] + 91.921;
   1:L PR[91] 10mm/sec FINE;
   1:  PR[GP1:91,1] = PR[GP1:90,1] + 118.737;
   1:  PR[GP1:91,2] = PR[GP1:90,2] + 92.750;
   1:L PR[91] 10mm/sec FINE;
   1:  PR[GP1:91,1] = PR[GP1:90,1] + 120.399;
   1:  PR[GP1:91,2] = PR[GP1:90,2] + 95.038;
   1:L PR[91] 10mm/sec FINE;
   1:  PR[GP1:91,1] = PR[GP1:90,1] + 121.182;
   1:  PR[GP1:91,2] = PR[GP1:90,2] + 96.573;
   1:L PR[91] 10mm/sec FINE;
   1:  PR[GP1:91,1] = PR[GP1:90,1] + 121.784;
   1:  PR[GP1:91,2] = PR[GP1:90,2] + 97.688;
   1:L PR[91] 10mm/sec FINE;
   1:  PR[GP1:91,1] = PR[GP1:90,1] + 122.495;
   1:  PR[GP1:91,2] = PR[GP1:90,2] + 99.615;
   1:L PR[91] 10mm/sec FINE;
   1:  PR[GP1:91,1] = PR[GP1:90,1] + 122.828;
   1:  PR[GP1:91,2] = PR[GP1:90,2] + 100.622;
   1:L PR[91] 10mm/sec FINE;
   1:  PR[GP1:91,1] = PR[GP1:90,1] + 123.073;
   1:  PR[GP1:91,2] = PR[GP1:90,2] + 101.819;
   1:L PR[91] 10mm/sec FINE;
   1:  PR[GP1:91,1] = PR[GP1:90,1] + 123.387;
   1:  PR[GP1:91,2] = PR[GP1:90,2] + 103.634;
   1:L PR[91] 10mm/sec FINE;
   1:  PR[GP1:91,1] = PR[GP1:90,1] + 123.424;
   1:  PR[GP1:91,2] = PR[GP1:90,2] + 105.531;
   1:L PR[91] 10mm/sec FINE;
   1:  PR[GP1:91,1] = PR[GP1:90,1] + 123.467;
   1:  PR[GP1:91,2] = PR[GP1:90,2] + 106.627;
   1:L PR[91] 10mm/sec FINE;
   1:  PR[GP1:91,1] = PR[GP1:90,1] + 122.976;
   1:  PR[GP1:91,2] = PR[GP1:90,2] + 110.329;
   1:L PR[91] 10mm/sec FINE;
   1:  PR[GP1:91,1] = PR[GP1:90,1] + 121.789;
   1:  PR[GP1:91,2] = PR[GP1:90,2] + 113.783;
   1:L PR[91] 10mm/sec FINE;
   1:  PR[GP1:91,1] = PR[GP1:90,1] + 119.980;
   1:  PR[GP1:91,2] = PR[GP1:90,2] + 116.854;
   1:L PR[91] 10mm/sec FINE;
   1:  PR[GP1:91,1] = PR[GP1:90,1] + 117.624;
   1:  PR[GP1:91,2] = PR[GP1:90,2] + 119.462;
   1:L PR[91] 10mm/sec FINE;
   1:  PR[GP1:91,1] = PR[GP1:90,1] + 114.847;
   1:  PR[GP1:91,2] = PR[GP1:90,2] + 121.519;
   1:L PR[91] 10mm/sec FINE;
   1:  PR[GP1:91,1] = PR[GP1:90,1] + 111.739;
   1:  PR[GP1:91,2] = PR[GP1:90,2] + 122.973;
   1:L PR[91] 10mm/sec FINE;
   1:  PR[GP1:91,1] = PR[GP1:90,1] + 108.374;
   1:  PR[GP1:91,2] = PR[GP1:90,2] + 123.796;
   1:L PR[91] 10mm/sec FINE;
   1:  PR[GP1:91,1] = PR[GP1:90,1] + 104.925;
   1:  PR[GP1:91,2] = PR[GP1:90,2] + 123.950;
   1:L PR[91] 10mm/sec FINE;
   1:  PR[GP1:91,1] = PR[GP1:90,1] + 101.599;
   1:  PR[GP1:91,2] = PR[GP1:90,2] + 123.489;
   1:L PR[91] 10mm/sec FINE;
   1:  PR[GP1:91,1] = PR[GP1:90,1] + 101.410;
   1:  PR[GP1:91,2] = PR[GP1:90,2] + 123.460;
   1:L PR[91] 10mm/sec FINE;
   1:  PR[GP1:91,1] = PR[GP1:90,1] + 98.165;
   1:  PR[GP1:91,2] = PR[GP1:90,2] + 122.336;
   1:L PR[91] 10mm/sec FINE;
   1:  PR[GP1:91,1] = PR[GP1:90,1] + 97.006;
   1:  PR[GP1:91,2] = PR[GP1:90,2] + 122.147;
   1:L PR[91] 10mm/sec FINE;
   1:  PR[GP1:91,1] = PR[GP1:90,1] + 96.572;
   1:  PR[GP1:91,2] = PR[GP1:90,2] + 122.245;
   1:L PR[91] 10mm/sec FINE;
   1:  PR[GP1:91,1] = PR[GP1:90,1] + 95.735;
   1:  PR[GP1:91,2] = PR[GP1:90,2] + 122.466;
   1:L PR[91] 10mm/sec FINE;
   1:  PR[GP1:91,1] = PR[GP1:90,1] + 94.062;
   1:  PR[GP1:91,2] = PR[GP1:90,2] + 122.852;
   1:L PR[91] 10mm/sec FINE;
   1:  PR[GP1:91,1] = PR[GP1:90,1] + 91.641;
   1:  PR[GP1:91,2] = PR[GP1:90,2] + 123.259;
   1:L PR[91] 10mm/sec FINE;
   1:  PR[GP1:91,1] = PR[GP1:90,1] + 89.827;
   1:  PR[GP1:91,2] = PR[GP1:90,2] + 123.492;
   1:L PR[91] 10mm/sec FINE;
   1:  PR[GP1:91,1] = PR[GP1:90,1] + 87.197;
   1:  PR[GP1:91,2] = PR[GP1:90,2] + 123.545;
   1:L PR[91] 10mm/sec FINE;
   1:  PR[GP1:91,1] = PR[GP1:90,1] + 86.334;
   1:  PR[GP1:91,2] = PR[GP1:90,2] + 123.549;
   1:L PR[91] 10mm/sec FINE;
   1:  PR[GP1:91,1] = PR[GP1:90,1] + 83.649;
   1:  PR[GP1:91,2] = PR[GP1:90,2] + 123.291;
   1:L PR[91] 10mm/sec FINE;
   1:  PR[GP1:91,1] = PR[GP1:90,1] + 83.430;
   1:  PR[GP1:91,2] = PR[GP1:90,2] + 123.266;
   1:L PR[91] 10mm/sec FINE;
   1:  PR[GP1:91,1] = PR[GP1:90,1] + 80.406;
   1:  PR[GP1:91,2] = PR[GP1:90,2] + 122.519;
   1:L PR[91] 10mm/sec FINE;
   1:  PR[GP1:91,1] = PR[GP1:90,1] + 78.862;
   1:  PR[GP1:91,2] = PR[GP1:90,2] + 121.930;
   1:L PR[91] 10mm/sec FINE;
   1:  PR[GP1:91,1] = PR[GP1:90,1] + 77.093;
   1:  PR[GP1:91,2] = PR[GP1:90,2] + 121.134;
   1:L PR[91] 10mm/sec FINE;
   1:  PR[GP1:91,1] = PR[GP1:90,1] + 76.158;
   1:  PR[GP1:91,2] = PR[GP1:90,2] + 120.624;
   1:L PR[91] 10mm/sec FINE;
   1:  PR[GP1:91,1] = PR[GP1:90,1] + 73.862;
   1:  PR[GP1:91,2] = PR[GP1:90,2] + 118.992;
   1:L PR[91] 10mm/sec FINE;
   1:  PR[GP1:91,1] = PR[GP1:90,1] + 73.464;
   1:  PR[GP1:91,2] = PR[GP1:90,2] + 118.690;
   1:L PR[91] 10mm/sec FINE;
   1:  PR[GP1:91,1] = PR[GP1:90,1] + 73.214;
   1:  PR[GP1:91,2] = PR[GP1:90,2] + 118.430;
   1:L PR[91] 10mm/sec FINE;
   1:  PR[GP1:91,1] = PR[GP1:90,1] + 71.113;
   1:  PR[GP1:91,2] = PR[GP1:90,2] + 116.105;
   1:L PR[91] 10mm/sec FINE;
   1:  PR[GP1:91,1] = PR[GP1:90,1] + 70.295;
   1:  PR[GP1:91,2] = PR[GP1:90,2] + 114.663;
   1:L PR[91] 10mm/sec FINE;
   1:  PR[GP1:91,1] = PR[GP1:90,1] + 69.447;
   1:  PR[GP1:91,2] = PR[GP1:90,2] + 113.099;
   1:L PR[91] 10mm/sec FINE;
   1:  PR[GP1:91,1] = PR[GP1:90,1] + 68.473;
   1:  PR[GP1:91,2] = PR[GP1:90,2] + 109.849;
   1:L PR[91] 10mm/sec FINE;
   1:  PR[GP1:91,1] = PR[GP1:90,1] + 68.456;
   1:  PR[GP1:91,2] = PR[GP1:90,2] + 109.635;
   1:L PR[91] 10mm/sec FINE;
   1:  PR[GP1:91,1] = PR[GP1:90,1] + 68.404;
   1:  PR[GP1:91,2] = PR[GP1:90,2] + 107.712;
   1:L PR[91] 10mm/sec FINE;
   1:  PR[GP1:91,1] = PR[GP1:90,1] + 68.387;
   1:  PR[GP1:91,2] = PR[GP1:90,2] + 106.397;
   1:L PR[91] 10mm/sec FINE;
   1:  PR[GP1:91,1] = PR[GP1:90,1] + 69.172;
   1:  PR[GP1:91,2] = PR[GP1:90,2] + 102.858;
   1:L PR[91] 10mm/sec FINE;
   1:  PR[GP1:91,1] = PR[GP1:90,1] + 69.376;
   1:  PR[GP1:91,2] = PR[GP1:90,2] + 102.355;
   1:L PR[91] 10mm/sec FINE;
   1:  PR[GP1:91,1] = PR[GP1:90,1] + 70.534;
   1:  PR[GP1:91,2] = PR[GP1:90,2] + 99.686;
   1:L PR[91] 10mm/sec FINE;
   1:  PR[GP1:91,1] = PR[GP1:90,1] + 71.149;
   1:  PR[GP1:91,2] = PR[GP1:90,2] + 98.709;
   1:L PR[91] 10mm/sec FINE;
   1:  PR[GP1:91,1] = PR[GP1:90,1] + 72.365;
   1:  PR[GP1:91,2] = PR[GP1:90,2] + 97.016;
   1:L PR[91] 10mm/sec FINE;
   1:  PR[GP1:91,1] = PR[GP1:90,1] + 73.676;
   1:  PR[GP1:91,2] = PR[GP1:90,2] + 95.522;
   1:L PR[91] 10mm/sec FINE;
   1:  PR[GP1:91,1] = PR[GP1:90,1] + 74.406;
   1:  PR[GP1:91,2] = PR[GP1:90,2] + 94.827;
   1:L PR[91] 10mm/sec FINE;
   1:  PR[GP1:91,1] = PR[GP1:90,1] + 74.811;
   1:  PR[GP1:91,2] = PR[GP1:90,2] + 94.908;
   1:  PR[GP1:91,3] = PR[GP1:90,3] + 39.900;
   1:L PR[91] 10mm/sec FINE;
   1:  PR[GP1:91,1] = PR[GP1:90,1] + 77.215;
   1:  PR[GP1:91,2] = PR[GP1:90,2] + 92.844;
   1:L PR[91] 10mm/sec FINE;
   1:  PR[GP1:91,1] = PR[GP1:90,1] + 77.848;
   1:  PR[GP1:91,2] = PR[GP1:90,2] + 92.412;
   1:L PR[91] 10mm/sec FINE;
   1:  PR[GP1:91,1] = PR[GP1:90,1] + 80.452;
   1:  PR[GP1:91,2] = PR[GP1:90,2] + 90.718;
   1:L PR[91] 10mm/sec FINE;
   1:  PR[GP1:91,1] = PR[GP1:90,1] + 82.391;
   1:  PR[GP1:91,2] = PR[GP1:90,2] + 89.775;
   1:L PR[91] 10mm/sec FINE;
   1:  PR[GP1:91,1] = PR[GP1:90,1] + 84.802;
   1:  PR[GP1:91,2] = PR[GP1:90,2] + 88.717;
   1:L PR[91] 10mm/sec FINE;
   1:  PR[GP1:91,1] = PR[GP1:90,1] + 86.215;
   1:  PR[GP1:91,2] = PR[GP1:90,2] + 88.226;
   1:L PR[91] 10mm/sec FINE;
   1:  PR[GP1:91,1] = PR[GP1:90,1] + 91.053;
   1:  PR[GP1:91,2] = PR[GP1:90,2] + 87.080;
   1:L PR[91] 10mm/sec FINE;
   1:  PR[GP1:91,1] = PR[GP1:90,1] + 92.871;
   1:  PR[GP1:91,2] = PR[GP1:90,2] + 86.974;
   1:L PR[91] 10mm/sec FINE;
   1:  PR[GP1:91,1] = PR[GP1:90,1] + 95.982;
   1:  PR[GP1:91,2] = PR[GP1:90,2] + 86.639;
   1:L PR[91] 10mm/sec FINE;
   1:  PR[GP1:91,1] = PR[GP1:90,1] + 96.933;
   1:  PR[GP1:91,2] = PR[GP1:90,2] + 86.599;
   1:L PR[91] 10mm/sec FINE;
   1:  PR[GP1:91,1] = PR[GP1:90,1] + 100.246;
   1:  PR[GP1:91,2] = PR[GP1:90,2] + 86.919;
   1:L PR[91] 10mm/sec FINE;
   1:  PR[GP1:91,1] = PR[GP1:90,1] + 101.138;
   1:  PR[GP1:91,2] = PR[GP1:90,2] + 86.864;
   1:L PR[91] 10mm/sec FINE;
   1:  PR[GP1:91,1] = PR[GP1:90,1] + 101.904;
   1:  PR[GP1:91,2] = PR[GP1:90,2] + 86.696;
   1:L PR[91] 10mm/sec FINE;
   1:  PR[GP1:91,1] = PR[GP1:90,1] + 104.086;
   1:  PR[GP1:91,2] = PR[GP1:90,2] + 86.369;
   1:L PR[91] 10mm/sec FINE;
   1:  PR[GP1:91,1] = PR[GP1:90,1] + 104.546;
   1:  PR[GP1:91,2] = PR[GP1:90,2] + 86.339;
   1:L PR[91] 10mm/sec FINE;
   1:  PR[GP1:91,1] = PR[GP1:90,1] + 106.959;
   1:  PR[GP1:91,2] = PR[GP1:90,2] + 86.358;
   1:L PR[91] 10mm/sec FINE;
   1:  PR[GP1:91,1] = PR[GP1:90,1] + 107.202;
   1:  PR[GP1:91,2] = PR[GP1:90,2] + 86.383;
   1:L PR[91] 10mm/sec FINE;
   1:  PR[GP1:91,1] = PR[GP1:90,1] + 109.738;
   1:  PR[GP1:91,2] = PR[GP1:90,2] + 86.808;
   1:L PR[91] 10mm/sec FINE;
   1:  PR[GP1:91,1] = PR[GP1:90,1] + 112.431;
   1:  PR[GP1:91,2] = PR[GP1:90,2] + 87.716;
   1:L PR[91] 10mm/sec FINE;
   1:  PR[GP1:91,1] = PR[GP1:90,1] + 114.817;
   1:  PR[GP1:91,2] = PR[GP1:90,2] + 88.965;
   1:L PR[91] 10mm/sec FINE;
   1:  PR[GP1:91,1] = PR[GP1:90,1] + 114.919;
   1:  PR[GP1:91,2] = PR[GP1:90,2] + 89.036;
   1:L PR[91] 10mm/sec FINE;
   1:  PR[GP1:91,1] = PR[GP1:90,1] + 117.013;
   1:  PR[GP1:91,2] = PR[GP1:90,2] + 90.596;
   1:L PR[91] 10mm/sec FINE;
   1:  PR[GP1:91,1] = PR[GP1:90,1] + 118.939;
   1:  PR[GP1:91,2] = PR[GP1:90,2] + 92.554;
   1:L PR[91] 10mm/sec FINE;
   1:  PR[GP1:91,1] = PR[GP1:90,1] + 120.558;
   1:  PR[GP1:91,2] = PR[GP1:90,2] + 94.813;
   1:L PR[91] 10mm/sec FINE;
   1:  PR[GP1:91,1] = PR[GP1:90,1] + 121.341;
   1:  PR[GP1:91,2] = PR[GP1:90,2] + 96.349;
   1:L PR[91] 10mm/sec FINE;
   1:  PR[GP1:91,1] = PR[GP1:90,1] + 121.844;
   1:  PR[GP1:91,2] = PR[GP1:90,2] + 97.349;
   1:L PR[91] 10mm/sec FINE;
   1:  PR[GP1:91,1] = PR[GP1:90,1] + 122.767;
   1:  PR[GP1:91,2] = PR[GP1:90,2] + 100.137;
   1:L PR[91] 10mm/sec FINE;
   1:  PR[GP1:91,1] = PR[GP1:90,1] + 123.232;
   1:  PR[GP1:91,2] = PR[GP1:90,2] + 102.439;
   1:L PR[91] 10mm/sec FINE;
   1:  PR[GP1:91,1] = PR[GP1:90,1] + 123.359;
   1:  PR[GP1:91,2] = PR[GP1:90,2] + 103.171;
   1:L PR[91] 10mm/sec FINE;
   1:  PR[GP1:91,1] = PR[GP1:90,1] + 123.428;
   1:  PR[GP1:91,2] = PR[GP1:90,2] + 106.215;
   1:L PR[91] 10mm/sec FINE;
   1:  PR[GP1:91,1] = PR[GP1:90,1] + 123.117;
   1:  PR[GP1:91,2] = PR[GP1:90,2] + 108.295;
   1:L PR[91] 10mm/sec FINE;
   1:  PR[GP1:91,1] = PR[GP1:90,1] + 122.899;
   1:  PR[GP1:91,2] = PR[GP1:90,2] + 109.977;
   1:L PR[91] 10mm/sec FINE;
   1:  PR[GP1:91,1] = PR[GP1:90,1] + 122.476;
   1:  PR[GP1:91,2] = PR[GP1:90,2] + 111.204;
   1:L PR[91] 10mm/sec FINE;
   1:  PR[GP1:91,1] = PR[GP1:90,1] + 121.731;
   1:  PR[GP1:91,2] = PR[GP1:90,2] + 113.459;
   1:L PR[91] 10mm/sec FINE;
   1:  PR[GP1:91,1] = PR[GP1:90,1] + 121.068;
   1:  PR[GP1:91,2] = PR[GP1:90,2] + 114.619;
   1:L PR[91] 10mm/sec FINE;
   1:  PR[GP1:91,1] = PR[GP1:90,1] + 119.917;
   1:  PR[GP1:91,2] = PR[GP1:90,2] + 116.562;
   1:L PR[91] 10mm/sec FINE;
   1:  PR[GP1:91,1] = PR[GP1:90,1] + 117.564;
   1:  PR[GP1:91,2] = PR[GP1:90,2] + 119.194;
   1:L PR[91] 10mm/sec FINE;
   1:  PR[GP1:91,1] = PR[GP1:90,1] + 114.774;
   1:  PR[GP1:91,2] = PR[GP1:90,2] + 121.276;
   1:L PR[91] 10mm/sec FINE;
   1:  PR[GP1:91,1] = PR[GP1:90,1] + 113.383;
   1:  PR[GP1:91,2] = PR[GP1:90,2] + 121.942;
   1:L PR[91] 10mm/sec FINE;
   1:  PR[GP1:91,1] = PR[GP1:90,1] + 111.645;
   1:  PR[GP1:91,2] = PR[GP1:90,2] + 122.752;
   1:L PR[91] 10mm/sec FINE;
   1:  PR[GP1:91,1] = PR[GP1:90,1] + 108.236;
   1:  PR[GP1:91,2] = PR[GP1:90,2] + 123.599;
   1:L PR[91] 10mm/sec FINE;
   1:  PR[GP1:91,1] = PR[GP1:90,1] + 104.835;
   1:  PR[GP1:91,2] = PR[GP1:90,2] + 123.752;
   1:L PR[91] 10mm/sec FINE;
   1:  PR[GP1:91,1] = PR[GP1:90,1] + 101.360;
   1:  PR[GP1:91,2] = PR[GP1:90,2] + 123.259;
   1:L PR[91] 10mm/sec FINE;
   1:  PR[GP1:91,1] = PR[GP1:90,1] + 100.488;
   1:  PR[GP1:91,2] = PR[GP1:90,2] + 122.995;
   1:L PR[91] 10mm/sec FINE;
   1:  PR[GP1:91,1] = PR[GP1:90,1] + 98.379;
   1:  PR[GP1:91,2] = PR[GP1:90,2] + 122.276;
   1:L PR[91] 10mm/sec FINE;
   1:  PR[GP1:91,1] = PR[GP1:90,1] + 97.212;
   1:  PR[GP1:91,2] = PR[GP1:90,2] + 122.111;
   1:L PR[91] 10mm/sec FINE;
   1:  PR[GP1:91,1] = PR[GP1:90,1] + 95.138;
   1:  PR[GP1:91,2] = PR[GP1:90,2] + 122.592;
   1:L PR[91] 10mm/sec FINE;
   1:  PR[GP1:91,1] = PR[GP1:90,1] + 92.181;
   1:  PR[GP1:91,2] = PR[GP1:90,2] + 123.089;
   1:L PR[91] 10mm/sec FINE;
   1:  PR[GP1:91,1] = PR[GP1:90,1] + 90.691;
   1:  PR[GP1:91,2] = PR[GP1:90,2] + 123.280;
   1:L PR[91] 10mm/sec FINE;
   1:  PR[GP1:91,1] = PR[GP1:90,1] + 88.530;
   1:  PR[GP1:91,2] = PR[GP1:90,2] + 123.324;
   1:L PR[91] 10mm/sec FINE;
   1:  PR[GP1:91,1] = PR[GP1:90,1] + 87.024;
   1:  PR[GP1:91,2] = PR[GP1:90,2] + 123.331;
   1:L PR[91] 10mm/sec FINE;
   1:  PR[GP1:91,1] = PR[GP1:90,1] + 84.432;
   1:  PR[GP1:91,2] = PR[GP1:90,2] + 123.082;
   1:L PR[91] 10mm/sec FINE;
   1:  PR[GP1:91,1] = PR[GP1:90,1] + 83.994;
   1:  PR[GP1:91,2] = PR[GP1:90,2] + 123.009;
   1:L PR[91] 10mm/sec FINE;
   1:  PR[GP1:91,1] = PR[GP1:90,1] + 82.320;
   1:  PR[GP1:91,2] = PR[GP1:90,2] + 122.646;
   1:L PR[91] 10mm/sec FINE;
   1:  PR[GP1:91,1] = PR[GP1:90,1] + 81.245;
   1:  PR[GP1:91,2] = PR[GP1:90,2] + 122.380;
   1:L PR[91] 10mm/sec FINE;
   1:  PR[GP1:91,1] = PR[GP1:90,1] + 79.239;
   1:  PR[GP1:91,2] = PR[GP1:90,2] + 121.615;
   1:L PR[91] 10mm/sec FINE;
   1:  PR[GP1:91,1] = PR[GP1:90,1] + 78.121;
   1:  PR[GP1:91,2] = PR[GP1:90,2] + 121.112;
   1:L PR[91] 10mm/sec FINE;
   1:  PR[GP1:91,1] = PR[GP1:90,1] + 76.712;
   1:  PR[GP1:91,2] = PR[GP1:90,2] + 120.342;
   1:L PR[91] 10mm/sec FINE;
   1:  PR[GP1:91,1] = PR[GP1:90,1] + 75.022;
   1:  PR[GP1:91,2] = PR[GP1:90,2] + 119.141;
   1:L PR[91] 10mm/sec FINE;
   1:  PR[GP1:91,1] = PR[GP1:90,1] + 74.177;
   1:  PR[GP1:91,2] = PR[GP1:90,2] + 118.501;
   1:L PR[91] 10mm/sec FINE;
   1:  PR[GP1:91,1] = PR[GP1:90,1] + 73.644;
   1:  PR[GP1:91,2] = PR[GP1:90,2] + 117.945;
   1:L PR[91] 10mm/sec FINE;
   1:  PR[GP1:91,1] = PR[GP1:90,1] + 71.933;
   1:  PR[GP1:91,2] = PR[GP1:90,2] + 116.051;
   1:L PR[91] 10mm/sec FINE;
   1:  PR[GP1:91,1] = PR[GP1:90,1] + 71.648;
   1:  PR[GP1:91,2] = PR[GP1:90,2] + 115.636;
   1:L PR[91] 10mm/sec FINE;
   1:  PR[GP1:91,1] = PR[GP1:90,1] + 70.238;
   1:  PR[GP1:91,2] = PR[GP1:90,2] + 113.122;
   1:L PR[91] 10mm/sec FINE;
   1:  PR[GP1:91,1] = PR[GP1:90,1] + 70.095;
   1:  PR[GP1:91,2] = PR[GP1:90,2] + 112.819;
   1:L PR[91] 10mm/sec FINE;
   1:  PR[GP1:91,1] = PR[GP1:90,1] + 69.158;
   1:  PR[GP1:91,2] = PR[GP1:90,2] + 109.696;
   1:L PR[91] 10mm/sec FINE;
   1:  PR[GP1:91,1] = PR[GP1:90,1] + 69.131;
   1:  PR[GP1:91,2] = PR[GP1:90,2] + 109.450;
   1:L PR[91] 10mm/sec FINE;
   1:  PR[GP1:91,1] = PR[GP1:90,1] + 69.084;
   1:  PR[GP1:91,2] = PR[GP1:90,2] + 106.526;
   1:L PR[91] 10mm/sec FINE;
   1:  PR[GP1:91,1] = PR[GP1:90,1] + 69.109;
   1:  PR[GP1:91,2] = PR[GP1:90,2] + 106.176;
   1:L PR[91] 10mm/sec FINE;
   1:  PR[GP1:91,1] = PR[GP1:90,1] + 69.674;
   1:  PR[GP1:91,2] = PR[GP1:90,2] + 103.616;
   1:L PR[91] 10mm/sec FINE;
   1:  PR[GP1:91,1] = PR[GP1:90,1] + 69.890;
   1:  PR[GP1:91,2] = PR[GP1:90,2] + 102.680;
   1:L PR[91] 10mm/sec FINE;
   1:  PR[GP1:91,1] = PR[GP1:90,1] + 70.326;
   1:  PR[GP1:91,2] = PR[GP1:90,2] + 101.602;
   1:L PR[91] 10mm/sec FINE;
   1:  PR[GP1:91,1] = PR[GP1:90,1] + 71.189;
   1:  PR[GP1:91,2] = PR[GP1:90,2] + 99.613;
   1:L PR[91] 10mm/sec FINE;
   1:  PR[GP1:91,1] = PR[GP1:90,1] + 72.122;
   1:  PR[GP1:91,2] = PR[GP1:90,2] + 98.130;
   1:L PR[91] 10mm/sec FINE;
   1:  PR[GP1:91,1] = PR[GP1:90,1] + 72.902;
   1:  PR[GP1:91,2] = PR[GP1:90,2] + 97.045;
   1:L PR[91] 10mm/sec FINE;
   1:  PR[GP1:91,1] = PR[GP1:90,1] + 74.607;
   1:  PR[GP1:91,2] = PR[GP1:90,2] + 95.102;
   1:L PR[91] 10mm/sec FINE;
   1:  PR[GP1:91,1] = PR[GP1:90,1] + 75.558;
   1:  PR[GP1:91,2] = PR[GP1:90,2] + 94.692;
   1:  PR[GP1:91,3] = PR[GP1:90,3] + 40.900;
   1:L PR[91] 10mm/sec FINE;
   1:  PR[GP1:91,1] = PR[GP1:90,1] + 77.904;
   1:  PR[GP1:91,2] = PR[GP1:90,2] + 92.676;
   1:L PR[91] 10mm/sec FINE;
   1:  PR[GP1:91,1] = PR[GP1:90,1] + 79.079;
   1:  PR[GP1:91,2] = PR[GP1:90,2] + 91.874;
   1:L PR[91] 10mm/sec FINE;
   1:  PR[GP1:91,1] = PR[GP1:90,1] + 81.282;
   1:  PR[GP1:91,2] = PR[GP1:90,2] + 90.441;
   1:L PR[91] 10mm/sec FINE;
   1:  PR[GP1:91,1] = PR[GP1:90,1] + 82.920;
   1:  PR[GP1:91,2] = PR[GP1:90,2] + 89.644;
   1:L PR[91] 10mm/sec FINE;
   1:  PR[GP1:91,1] = PR[GP1:90,1] + 85.846;
   1:  PR[GP1:91,2] = PR[GP1:90,2] + 88.360;
   1:L PR[91] 10mm/sec FINE;
   1:  PR[GP1:91,1] = PR[GP1:90,1] + 86.873;
   1:  PR[GP1:91,2] = PR[GP1:90,2] + 88.004;
   1:L PR[91] 10mm/sec FINE;
   1:  PR[GP1:91,1] = PR[GP1:90,1] + 91.675;
   1:  PR[GP1:91,2] = PR[GP1:90,2] + 86.855;
   1:L PR[91] 10mm/sec FINE;
   1:  PR[GP1:91,1] = PR[GP1:90,1] + 91.921;
   1:  PR[GP1:91,2] = PR[GP1:90,2] + 86.786;
   1:L PR[91] 10mm/sec FINE;
   1:  PR[GP1:91,1] = PR[GP1:90,1] + 96.477;
   1:  PR[GP1:91,2] = PR[GP1:90,2] + 86.295;
   1:L PR[91] 10mm/sec FINE;
   1:  PR[GP1:91,1] = PR[GP1:90,1] + 97.969;
   1:  PR[GP1:91,2] = PR[GP1:90,2] + 86.233;
   1:L PR[91] 10mm/sec FINE;
   1:  PR[GP1:91,1] = PR[GP1:90,1] + 98.558;
   1:  PR[GP1:91,2] = PR[GP1:90,2] + 86.303;
   1:L PR[91] 10mm/sec FINE;
   1:  PR[GP1:91,1] = PR[GP1:90,1] + 100.745;
   1:  PR[GP1:91,2] = PR[GP1:90,2] + 86.512;
   1:L PR[91] 10mm/sec FINE;
   1:  PR[GP1:91,1] = PR[GP1:90,1] + 101.566;
   1:  PR[GP1:91,2] = PR[GP1:90,2] + 86.462;
   1:L PR[91] 10mm/sec FINE;
   1:  PR[GP1:91,1] = PR[GP1:90,1] + 104.314;
   1:  PR[GP1:91,2] = PR[GP1:90,2] + 86.032;
   1:L PR[91] 10mm/sec FINE;
   1:  PR[GP1:91,1] = PR[GP1:90,1] + 104.523;
   1:  PR[GP1:91,2] = PR[GP1:90,2] + 86.016;
   1:L PR[91] 10mm/sec FINE;
   1:  PR[GP1:91,1] = PR[GP1:90,1] + 107.012;
   1:  PR[GP1:91,2] = PR[GP1:90,2] + 86.018;
   1:L PR[91] 10mm/sec FINE;
   1:  PR[GP1:91,1] = PR[GP1:90,1] + 107.475;
   1:  PR[GP1:91,2] = PR[GP1:90,2] + 86.058;
   1:L PR[91] 10mm/sec FINE;
   1:  PR[GP1:91,1] = PR[GP1:90,1] + 109.697;
   1:  PR[GP1:91,2] = PR[GP1:90,2] + 86.417;
   1:L PR[91] 10mm/sec FINE;
   1:  PR[GP1:91,1] = PR[GP1:90,1] + 110.334;
   1:  PR[GP1:91,2] = PR[GP1:90,2] + 86.581;
   1:L PR[91] 10mm/sec FINE;
   1:  PR[GP1:91,1] = PR[GP1:90,1] + 112.314;
   1:  PR[GP1:91,2] = PR[GP1:90,2] + 87.242;
   1:L PR[91] 10mm/sec FINE;
   1:  PR[GP1:91,1] = PR[GP1:90,1] + 113.010;
   1:  PR[GP1:91,2] = PR[GP1:90,2] + 87.551;
   1:L PR[91] 10mm/sec FINE;
   1:  PR[GP1:91,1] = PR[GP1:90,1] + 114.797;
   1:  PR[GP1:91,2] = PR[GP1:90,2] + 88.492;
   1:L PR[91] 10mm/sec FINE;
   1:  PR[GP1:91,1] = PR[GP1:90,1] + 115.425;
   1:  PR[GP1:91,2] = PR[GP1:90,2] + 88.909;
   1:L PR[91] 10mm/sec FINE;
   1:  PR[GP1:91,1] = PR[GP1:90,1] + 117.076;
   1:  PR[GP1:91,2] = PR[GP1:90,2] + 90.162;
   1:L PR[91] 10mm/sec FINE;
   1:  PR[GP1:91,1] = PR[GP1:90,1] + 117.522;
   1:  PR[GP1:91,2] = PR[GP1:90,2] + 90.580;
   1:L PR[91] 10mm/sec FINE;
   1:  PR[GP1:91,1] = PR[GP1:90,1] + 119.076;
   1:  PR[GP1:91,2] = PR[GP1:90,2] + 92.220;
   1:L PR[91] 10mm/sec FINE;
   1:  PR[GP1:91,1] = PR[GP1:90,1] + 119.273;
   1:  PR[GP1:91,2] = PR[GP1:90,2] + 92.479;
   1:L PR[91] 10mm/sec FINE;
   1:  PR[GP1:91,1] = PR[GP1:90,1] + 120.715;
   1:  PR[GP1:91,2] = PR[GP1:90,2] + 94.586;
   1:L PR[91] 10mm/sec FINE;
   1:  PR[GP1:91,1] = PR[GP1:90,1] + 121.970;
   1:  PR[GP1:91,2] = PR[GP1:90,2] + 97.078;
   1:L PR[91] 10mm/sec FINE;
   1:  PR[GP1:91,1] = PR[GP1:90,1] + 122.873;
   1:  PR[GP1:91,2] = PR[GP1:90,2] + 99.802;
   1:L PR[91] 10mm/sec FINE;
   1:  PR[GP1:91,1] = PR[GP1:90,1] + 123.371;
   1:  PR[GP1:91,2] = PR[GP1:90,2] + 102.726;
   1:L PR[91] 10mm/sec FINE;
   1:  PR[GP1:91,1] = PR[GP1:90,1] + 123.378;
   1:  PR[GP1:91,2] = PR[GP1:90,2] + 104.004;
   1:L PR[91] 10mm/sec FINE;
   1:  PR[GP1:91,1] = PR[GP1:90,1] + 123.417;
   1:  PR[GP1:91,2] = PR[GP1:90,2] + 105.791;
   1:L PR[91] 10mm/sec FINE;
   1:  PR[GP1:91,1] = PR[GP1:90,1] + 122.870;
   1:  PR[GP1:91,2] = PR[GP1:90,2] + 109.605;
   1:L PR[91] 10mm/sec FINE;
   1:  PR[GP1:91,1] = PR[GP1:90,1] + 122.299;
   1:  PR[GP1:91,2] = PR[GP1:90,2] + 111.241;
   1:L PR[91] 10mm/sec FINE;
   1:  PR[GP1:91,1] = PR[GP1:90,1] + 121.674;
   1:  PR[GP1:91,2] = PR[GP1:90,2] + 113.133;
   1:L PR[91] 10mm/sec FINE;
   1:  PR[GP1:91,1] = PR[GP1:90,1] + 120.423;
   1:  PR[GP1:91,2] = PR[GP1:90,2] + 115.323;
   1:L PR[91] 10mm/sec FINE;
   1:  PR[GP1:91,1] = PR[GP1:90,1] + 119.864;
   1:  PR[GP1:91,2] = PR[GP1:90,2] + 116.267;
   1:L PR[91] 10mm/sec FINE;
   1:  PR[GP1:91,1] = PR[GP1:90,1] + 118.412;
   1:  PR[GP1:91,2] = PR[GP1:90,2] + 117.918;
   1:L PR[91] 10mm/sec FINE;
   1:  PR[GP1:91,1] = PR[GP1:90,1] + 117.504;
   1:  PR[GP1:91,2] = PR[GP1:90,2] + 118.926;
   1:L PR[91] 10mm/sec FINE;
   1:  PR[GP1:91,1] = PR[GP1:90,1] + 114.703;
   1:  PR[GP1:91,2] = PR[GP1:90,2] + 121.032;
   1:L PR[91] 10mm/sec FINE;
   1:  PR[GP1:91,1] = PR[GP1:90,1] + 111.551;
   1:  PR[GP1:91,2] = PR[GP1:90,2] + 122.532;
   1:L PR[91] 10mm/sec FINE;
   1:  PR[GP1:91,1] = PR[GP1:90,1] + 108.178;
   1:  PR[GP1:91,2] = PR[GP1:90,2] + 123.382;
   1:L PR[91] 10mm/sec FINE;
   1:  PR[GP1:91,1] = PR[GP1:90,1] + 106.784;
   1:  PR[GP1:91,2] = PR[GP1:90,2] + 123.462;
   1:L PR[91] 10mm/sec FINE;
   1:  PR[GP1:91,1] = PR[GP1:90,1] + 104.745;
   1:  PR[GP1:91,2] = PR[GP1:90,2] + 123.554;
   1:L PR[91] 10mm/sec FINE;
   1:  PR[GP1:91,1] = PR[GP1:90,1] + 101.332;
   1:  PR[GP1:91,2] = PR[GP1:90,2] + 123.056;
   1:L PR[91] 10mm/sec FINE;
   1:  PR[GP1:91,1] = PR[GP1:90,1] + 100.198;
   1:  PR[GP1:91,2] = PR[GP1:90,2] + 122.724;
   1:L PR[91] 10mm/sec FINE;
   1:  PR[GP1:91,1] = PR[GP1:90,1] + 98.600;
   1:  PR[GP1:91,2] = PR[GP1:90,2] + 122.202;
   1:L PR[91] 10mm/sec FINE;
   1:  PR[GP1:91,1] = PR[GP1:90,1] + 97.431;
   1:  PR[GP1:91,2] = PR[GP1:90,2] + 122.058;
   1:L PR[91] 10mm/sec FINE;
   1:  PR[GP1:91,1] = PR[GP1:90,1] + 96.214;
   1:  PR[GP1:91,2] = PR[GP1:90,2] + 122.332;
   1:L PR[91] 10mm/sec FINE;
   1:  PR[GP1:91,1] = PR[GP1:90,1] + 92.721;
   1:  PR[GP1:91,2] = PR[GP1:90,2] + 122.919;
   1:L PR[91] 10mm/sec FINE;
   1:  PR[GP1:91,1] = PR[GP1:90,1] + 91.556;
   1:  PR[GP1:91,2] = PR[GP1:90,2] + 123.069;
   1:L PR[91] 10mm/sec FINE;
   1:  PR[GP1:91,1] = PR[GP1:90,1] + 89.864;
   1:  PR[GP1:91,2] = PR[GP1:90,2] + 123.103;
   1:L PR[91] 10mm/sec FINE;
   1:  PR[GP1:91,1] = PR[GP1:90,1] + 87.714;
   1:  PR[GP1:91,2] = PR[GP1:90,2] + 123.113;
   1:L PR[91] 10mm/sec FINE;
   1:  PR[GP1:91,1] = PR[GP1:90,1] + 85.498;
   1:  PR[GP1:91,2] = PR[GP1:90,2] + 122.900;
   1:L PR[91] 10mm/sec FINE;
   1:  PR[GP1:91,1] = PR[GP1:90,1] + 84.546;
   1:  PR[GP1:91,2] = PR[GP1:90,2] + 122.742;
   1:L PR[91] 10mm/sec FINE;
   1:  PR[GP1:91,1] = PR[GP1:90,1] + 82.090;
   1:  PR[GP1:91,2] = PR[GP1:90,2] + 122.208;
   1:L PR[91] 10mm/sec FINE;
   1:  PR[GP1:91,1] = PR[GP1:90,1] + 80.943;
   1:  PR[GP1:91,2] = PR[GP1:90,2] + 121.805;
   1:L PR[91] 10mm/sec FINE;
   1:  PR[GP1:91,1] = PR[GP1:90,1] + 79.615;
   1:  PR[GP1:91,2] = PR[GP1:90,2] + 121.299;
   1:L PR[91] 10mm/sec FINE;
   1:  PR[GP1:91,1] = PR[GP1:90,1] + 79.149;
   1:  PR[GP1:91,2] = PR[GP1:90,2] + 121.089;
   1:L PR[91] 10mm/sec FINE;
   1:  PR[GP1:91,1] = PR[GP1:90,1] + 77.266;
   1:  PR[GP1:91,2] = PR[GP1:90,2] + 120.061;
   1:L PR[91] 10mm/sec FINE;
   1:  PR[GP1:91,1] = PR[GP1:90,1] + 76.183;
   1:  PR[GP1:91,2] = PR[GP1:90,2] + 119.291;
   1:L PR[91] 10mm/sec FINE;
   1:  PR[GP1:91,1] = PR[GP1:90,1] + 74.891;
   1:  PR[GP1:91,2] = PR[GP1:90,2] + 118.313;
   1:L PR[91] 10mm/sec FINE;
   1:  PR[GP1:91,1] = PR[GP1:90,1] + 74.074;
   1:  PR[GP1:91,2] = PR[GP1:90,2] + 117.460;
   1:L PR[91] 10mm/sec FINE;
   1:  PR[GP1:91,1] = PR[GP1:90,1] + 72.758;
   1:  PR[GP1:91,2] = PR[GP1:90,2] + 116.003;
   1:L PR[91] 10mm/sec FINE;
   1:  PR[GP1:91,1] = PR[GP1:90,1] + 72.223;
   1:  PR[GP1:91,2] = PR[GP1:90,2] + 115.222;
   1:L PR[91] 10mm/sec FINE;
   1:  PR[GP1:91,1] = PR[GP1:90,1] + 71.106;
   1:  PR[GP1:91,2] = PR[GP1:90,2] + 113.231;
   1:L PR[91] 10mm/sec FINE;
   1:  PR[GP1:91,1] = PR[GP1:90,1] + 70.772;
   1:  PR[GP1:91,2] = PR[GP1:90,2] + 112.522;
   1:L PR[91] 10mm/sec FINE;
   1:  PR[GP1:91,1] = PR[GP1:90,1] + 69.891;
   1:  PR[GP1:91,2] = PR[GP1:90,2] + 109.568;
   1:L PR[91] 10mm/sec FINE;
   1:  PR[GP1:91,1] = PR[GP1:90,1] + 69.822;
   1:  PR[GP1:91,2] = PR[GP1:90,2] + 108.956;
   1:L PR[91] 10mm/sec FINE;
   1:  PR[GP1:91,1] = PR[GP1:90,1] + 69.784;
   1:  PR[GP1:91,2] = PR[GP1:90,2] + 106.621;
   1:L PR[91] 10mm/sec FINE;
   1:  PR[GP1:91,1] = PR[GP1:90,1] + 69.834;
   1:  PR[GP1:91,2] = PR[GP1:90,2] + 105.946;
   1:L PR[91] 10mm/sec FINE;
   1:  PR[GP1:91,1] = PR[GP1:90,1] + 70.277;
   1:  PR[GP1:91,2] = PR[GP1:90,2] + 103.936;
   1:L PR[91] 10mm/sec FINE;
   1:  PR[GP1:91,1] = PR[GP1:90,1] + 70.608;
   1:  PR[GP1:91,2] = PR[GP1:90,2] + 102.501;
   1:L PR[91] 10mm/sec FINE;
   1:  PR[GP1:91,1] = PR[GP1:90,1] + 71.277;
   1:  PR[GP1:91,2] = PR[GP1:90,2] + 100.848;
   1:L PR[91] 10mm/sec FINE;
   1:  PR[GP1:91,1] = PR[GP1:90,1] + 71.844;
   1:  PR[GP1:91,2] = PR[GP1:90,2] + 99.541;
   1:L PR[91] 10mm/sec FINE;
   1:  PR[GP1:91,1] = PR[GP1:90,1] + 73.096;
   1:  PR[GP1:91,2] = PR[GP1:90,2] + 97.551;
   1:L PR[91] 10mm/sec FINE;
   1:  PR[GP1:91,1] = PR[GP1:90,1] + 73.439;
   1:  PR[GP1:91,2] = PR[GP1:90,2] + 97.073;
   1:L PR[91] 10mm/sec FINE;
   1:  PR[GP1:91,1] = PR[GP1:90,1] + 75.353;
   1:  PR[GP1:91,2] = PR[GP1:90,2] + 94.902;
   1:L PR[91] 10mm/sec FINE;
   1:  PR[GP1:91,1] = PR[GP1:90,1] + 76.537;
   1:  PR[GP1:91,2] = PR[GP1:90,2] + 94.275;
   1:  PR[GP1:91,3] = PR[GP1:90,3] + 41.900;
   1:L PR[91] 10mm/sec FINE;
   1:  PR[GP1:91,1] = PR[GP1:90,1] + 78.593;
   1:  PR[GP1:91,2] = PR[GP1:90,2] + 92.508;
   1:L PR[91] 10mm/sec FINE;
   1:  PR[GP1:91,1] = PR[GP1:90,1] + 80.311;
   1:  PR[GP1:91,2] = PR[GP1:90,2] + 91.336;
   1:L PR[91] 10mm/sec FINE;
   1:  PR[GP1:91,1] = PR[GP1:90,1] + 82.112;
   1:  PR[GP1:91,2] = PR[GP1:90,2] + 90.164;
   1:L PR[91] 10mm/sec FINE;
   1:  PR[GP1:91,1] = PR[GP1:90,1] + 83.450;
   1:  PR[GP1:91,2] = PR[GP1:90,2] + 89.513;
   1:L PR[91] 10mm/sec FINE;
   1:  PR[GP1:91,1] = PR[GP1:90,1] + 86.890;
   1:  PR[GP1:91,2] = PR[GP1:90,2] + 88.004;
   1:L PR[91] 10mm/sec FINE;
   1:  PR[GP1:91,1] = PR[GP1:90,1] + 87.530;
   1:  PR[GP1:91,2] = PR[GP1:90,2] + 87.782;
   1:L PR[91] 10mm/sec FINE;
   1:  PR[GP1:91,1] = PR[GP1:90,1] + 90.554;
   1:  PR[GP1:91,2] = PR[GP1:90,2] + 87.059;
   1:L PR[91] 10mm/sec FINE;
   1:  PR[GP1:91,1] = PR[GP1:90,1] + 92.351;
   1:  PR[GP1:91,2] = PR[GP1:90,2] + 86.524;
   1:L PR[91] 10mm/sec FINE;
   1:  PR[GP1:91,1] = PR[GP1:90,1] + 92.933;
   1:  PR[GP1:91,2] = PR[GP1:90,2] + 86.387;
   1:L PR[91] 10mm/sec FINE;
   1:  PR[GP1:91,1] = PR[GP1:90,1] + 96.972;
   1:  PR[GP1:91,2] = PR[GP1:90,2] + 85.952;
   1:L PR[91] 10mm/sec FINE;
   1:  PR[GP1:91,1] = PR[GP1:90,1] + 99.007;
   1:  PR[GP1:91,2] = PR[GP1:90,2] + 85.867;
   1:L PR[91] 10mm/sec FINE;
   1:  PR[GP1:91,1] = PR[GP1:90,1] + 99.812;
   1:  PR[GP1:91,2] = PR[GP1:90,2] + 85.963;
   1:L PR[91] 10mm/sec FINE;
   1:  PR[GP1:91,1] = PR[GP1:90,1] + 101.267;
   1:  PR[GP1:91,2] = PR[GP1:90,2] + 86.105;
   1:L PR[91] 10mm/sec FINE;
   1:  PR[GP1:91,1] = PR[GP1:90,1] + 102.025;
   1:  PR[GP1:91,2] = PR[GP1:90,2] + 86.059;
   1:L PR[91] 10mm/sec FINE;
   1:  PR[GP1:91,1] = PR[GP1:90,1] + 104.198;
   1:  PR[GP1:91,2] = PR[GP1:90,2] + 85.723;
   1:L PR[91] 10mm/sec FINE;
   1:  PR[GP1:91,1] = PR[GP1:90,1] + 105.076;
   1:  PR[GP1:91,2] = PR[GP1:90,2] + 85.656;
   1:L PR[91] 10mm/sec FINE;
   1:  PR[GP1:91,1] = PR[GP1:90,1] + 106.894;
   1:  PR[GP1:91,2] = PR[GP1:90,2] + 85.658;
   1:L PR[91] 10mm/sec FINE;
   1:  PR[GP1:91,1] = PR[GP1:90,1] + 108.076;
   1:  PR[GP1:91,2] = PR[GP1:90,2] + 85.760;
   1:L PR[91] 10mm/sec FINE;
   1:  PR[GP1:91,1] = PR[GP1:90,1] + 109.586;
   1:  PR[GP1:91,2] = PR[GP1:90,2] + 86.004;
   1:L PR[91] 10mm/sec FINE;
   1:  PR[GP1:91,1] = PR[GP1:90,1] + 110.973;
   1:  PR[GP1:91,2] = PR[GP1:90,2] + 86.360;
   1:L PR[91] 10mm/sec FINE;
   1:  PR[GP1:91,1] = PR[GP1:90,1] + 112.218;
   1:  PR[GP1:91,2] = PR[GP1:90,2] + 86.776;
   1:L PR[91] 10mm/sec FINE;
   1:  PR[GP1:91,1] = PR[GP1:90,1] + 113.674;
   1:  PR[GP1:91,2] = PR[GP1:90,2] + 87.422;
   1:L PR[91] 10mm/sec FINE;
   1:  PR[GP1:91,1] = PR[GP1:90,1] + 114.728;
   1:  PR[GP1:91,2] = PR[GP1:90,2] + 87.978;
   1:L PR[91] 10mm/sec FINE;
   1:  PR[GP1:91,1] = PR[GP1:90,1] + 116.094;
   1:  PR[GP1:91,2] = PR[GP1:90,2] + 88.883;
   1:L PR[91] 10mm/sec FINE;
   1:  PR[GP1:91,1] = PR[GP1:90,1] + 117.045;
   1:  PR[GP1:91,2] = PR[GP1:90,2] + 89.605;
   1:L PR[91] 10mm/sec FINE;
   1:  PR[GP1:91,1] = PR[GP1:90,1] + 118.170;
   1:  PR[GP1:91,2] = PR[GP1:90,2] + 90.660;
   1:L PR[91] 10mm/sec FINE;
   1:  PR[GP1:91,1] = PR[GP1:90,1] + 119.093;
   1:  PR[GP1:91,2] = PR[GP1:90,2] + 91.633;
   1:L PR[91] 10mm/sec FINE;
   1:  PR[GP1:91,1] = PR[GP1:90,1] + 119.874;
   1:  PR[GP1:91,2] = PR[GP1:90,2] + 92.660;
   1:L PR[91] 10mm/sec FINE;
   1:  PR[GP1:91,1] = PR[GP1:90,1] + 120.795;
   1:  PR[GP1:91,2] = PR[GP1:90,2] + 94.019;
   1:L PR[91] 10mm/sec FINE;
   1:  PR[GP1:91,1] = PR[GP1:90,1] + 121.209;
   1:  PR[GP1:91,2] = PR[GP1:90,2] + 94.801;
   1:L PR[91] 10mm/sec FINE;
   1:  PR[GP1:91,1] = PR[GP1:90,1] + 122.095;
   1:  PR[GP1:91,2] = PR[GP1:90,2] + 96.685;
   1:L PR[91] 10mm/sec FINE;
   1:  PR[GP1:91,1] = PR[GP1:90,1] + 122.210;
   1:  PR[GP1:91,2] = PR[GP1:90,2] + 97.017;
   1:L PR[91] 10mm/sec FINE;
   1:  PR[GP1:91,1] = PR[GP1:90,1] + 122.614;
   1:  PR[GP1:91,2] = PR[GP1:90,2] + 98.367;
   1:L PR[91] 10mm/sec FINE;
   1:  PR[GP1:91,1] = PR[GP1:90,1] + 122.981;
   1:  PR[GP1:91,2] = PR[GP1:90,2] + 99.471;
   1:L PR[91] 10mm/sec FINE;
   1:  PR[GP1:91,1] = PR[GP1:90,1] + 123.478;
   1:  PR[GP1:91,2] = PR[GP1:90,2] + 102.328;
   1:L PR[91] 10mm/sec FINE;
   1:  PR[GP1:91,1] = PR[GP1:90,1] + 123.494;
   1:  PR[GP1:91,2] = PR[GP1:90,2] + 105.342;
   1:L PR[91] 10mm/sec FINE;
   1:  PR[GP1:91,1] = PR[GP1:90,1] + 123.241;
   1:  PR[GP1:91,2] = PR[GP1:90,2] + 106.946;
   1:L PR[91] 10mm/sec FINE;
   1:  PR[GP1:91,1] = PR[GP1:90,1] + 122.922;
   1:  PR[GP1:91,2] = PR[GP1:90,2] + 109.201;
   1:L PR[91] 10mm/sec FINE;
   1:  PR[GP1:91,1] = PR[GP1:90,1] + 122.188;
   1:  PR[GP1:91,2] = PR[GP1:90,2] + 111.306;
   1:L PR[91] 10mm/sec FINE;
   1:  PR[GP1:91,1] = PR[GP1:90,1] + 121.692;
   1:  PR[GP1:91,2] = PR[GP1:90,2] + 112.779;
   1:L PR[91] 10mm/sec FINE;
   1:  PR[GP1:91,1] = PR[GP1:90,1] + 119.816;
   1:  PR[GP1:91,2] = PR[GP1:90,2] + 115.969;
   1:L PR[91] 10mm/sec FINE;
   1:  PR[GP1:91,1] = PR[GP1:90,1] + 117.443;
   1:  PR[GP1:91,2] = PR[GP1:90,2] + 118.659;
   1:L PR[91] 10mm/sec FINE;
   1:  PR[GP1:91,1] = PR[GP1:90,1] + 114.630;
   1:  PR[GP1:91,2] = PR[GP1:90,2] + 120.789;
   1:L PR[91] 10mm/sec FINE;
   1:  PR[GP1:91,1] = PR[GP1:90,1] + 111.483;
   1:  PR[GP1:91,2] = PR[GP1:90,2] + 122.304;
   1:L PR[91] 10mm/sec FINE;
   1:  PR[GP1:91,1] = PR[GP1:90,1] + 108.173;
   1:  PR[GP1:91,2] = PR[GP1:90,2] + 123.151;
   1:L PR[91] 10mm/sec FINE;
   1:  PR[GP1:91,1] = PR[GP1:90,1] + 104.665;
   1:  PR[GP1:91,2] = PR[GP1:90,2] + 123.354;
   1:L PR[91] 10mm/sec FINE;
   1:  PR[GP1:91,1] = PR[GP1:90,1] + 101.304;
   1:  PR[GP1:91,2] = PR[GP1:90,2] + 122.853;
   1:L PR[91] 10mm/sec FINE;
   1:  PR[GP1:91,1] = PR[GP1:90,1] + 99.554;
   1:  PR[GP1:91,2] = PR[GP1:90,2] + 122.341;
   1:L PR[91] 10mm/sec FINE;
   1:  PR[GP1:91,1] = PR[GP1:90,1] + 98.833;
   1:  PR[GP1:91,2] = PR[GP1:90,2] + 122.112;
   1:L PR[91] 10mm/sec FINE;
   1:  PR[GP1:91,1] = PR[GP1:90,1] + 97.661;
   1:  PR[GP1:91,2] = PR[GP1:90,2] + 121.984;
   1:L PR[91] 10mm/sec FINE;
   1:  PR[GP1:91,1] = PR[GP1:90,1] + 97.289;
   1:  PR[GP1:91,2] = PR[GP1:90,2] + 122.072;
   1:L PR[91] 10mm/sec FINE;
   1:  PR[GP1:91,1] = PR[GP1:90,1] + 93.261;
   1:  PR[GP1:91,2] = PR[GP1:90,2] + 122.749;
   1:L PR[91] 10mm/sec FINE;
   1:  PR[GP1:91,1] = PR[GP1:90,1] + 92.420;
   1:  PR[GP1:91,2] = PR[GP1:90,2] + 122.857;
   1:L PR[91] 10mm/sec FINE;
   1:  PR[GP1:91,1] = PR[GP1:90,1] + 91.197;
   1:  PR[GP1:91,2] = PR[GP1:90,2] + 122.882;
   1:L PR[91] 10mm/sec FINE;
   1:  PR[GP1:91,1] = PR[GP1:90,1] + 88.404;
   1:  PR[GP1:91,2] = PR[GP1:90,2] + 122.895;
   1:L PR[91] 10mm/sec FINE;
   1:  PR[GP1:91,1] = PR[GP1:90,1] + 86.563;
   1:  PR[GP1:91,2] = PR[GP1:90,2] + 122.718;
   1:L PR[91] 10mm/sec FINE;
   1:  PR[GP1:91,1] = PR[GP1:90,1] + 85.099;
   1:  PR[GP1:91,2] = PR[GP1:90,2] + 122.475;
   1:L PR[91] 10mm/sec FINE;
   1:  PR[GP1:91,1] = PR[GP1:90,1] + 82.951;
   1:  PR[GP1:91,2] = PR[GP1:90,2] + 122.008;
   1:L PR[91] 10mm/sec FINE;
   1:  PR[GP1:91,1] = PR[GP1:90,1] + 80.084;
   1:  PR[GP1:91,2] = PR[GP1:90,2] + 120.998;
   1:L PR[91] 10mm/sec FINE;
   1:  PR[GP1:91,1] = PR[GP1:90,1] + 79.498;
   1:  PR[GP1:91,2] = PR[GP1:90,2] + 120.696;
   1:L PR[91] 10mm/sec FINE;
   1:  PR[GP1:91,1] = PR[GP1:90,1] + 77.820;
   1:  PR[GP1:91,2] = PR[GP1:90,2] + 119.779;
   1:L PR[91] 10mm/sec FINE;
   1:  PR[GP1:91,1] = PR[GP1:90,1] + 77.343;
   1:  PR[GP1:91,2] = PR[GP1:90,2] + 119.440;
   1:L PR[91] 10mm/sec FINE;
   1:  PR[GP1:91,1] = PR[GP1:90,1] + 75.605;
   1:  PR[GP1:91,2] = PR[GP1:90,2] + 118.124;
   1:L PR[91] 10mm/sec FINE;
   1:  PR[GP1:91,1] = PR[GP1:90,1] + 74.505;
   1:  PR[GP1:91,2] = PR[GP1:90,2] + 116.976;
   1:L PR[91] 10mm/sec FINE;
   1:  PR[GP1:91,1] = PR[GP1:90,1] + 73.583;
   1:  PR[GP1:91,2] = PR[GP1:90,2] + 115.956;
   1:L PR[91] 10mm/sec FINE;
   1:  PR[GP1:91,1] = PR[GP1:90,1] + 72.798;
   1:  PR[GP1:91,2] = PR[GP1:90,2] + 114.808;
   1:L PR[91] 10mm/sec FINE;
   1:  PR[GP1:91,1] = PR[GP1:90,1] + 71.974;
   1:  PR[GP1:91,2] = PR[GP1:90,2] + 113.340;
   1:L PR[91] 10mm/sec FINE;
   1:  PR[GP1:91,1] = PR[GP1:90,1] + 71.450;
   1:  PR[GP1:91,2] = PR[GP1:90,2] + 112.225;
   1:L PR[91] 10mm/sec FINE;
   1:  PR[GP1:91,1] = PR[GP1:90,1] + 70.623;
   1:  PR[GP1:91,2] = PR[GP1:90,2] + 109.441;
   1:L PR[91] 10mm/sec FINE;
   1:  PR[GP1:91,1] = PR[GP1:90,1] + 70.513;
   1:  PR[GP1:91,2] = PR[GP1:90,2] + 108.462;
   1:L PR[91] 10mm/sec FINE;
   1:  PR[GP1:91,1] = PR[GP1:90,1] + 70.485;
   1:  PR[GP1:91,2] = PR[GP1:90,2] + 106.715;
   1:L PR[91] 10mm/sec FINE;
   1:  PR[GP1:91,1] = PR[GP1:90,1] + 70.558;
   1:  PR[GP1:91,2] = PR[GP1:90,2] + 105.716;
   1:L PR[91] 10mm/sec FINE;
   1:  PR[GP1:91,1] = PR[GP1:90,1] + 70.880;
   1:  PR[GP1:91,2] = PR[GP1:90,2] + 104.257;
   1:L PR[91] 10mm/sec FINE;
   1:  PR[GP1:91,1] = PR[GP1:90,1] + 71.326;
   1:  PR[GP1:91,2] = PR[GP1:90,2] + 102.322;
   1:L PR[91] 10mm/sec FINE;
   1:  PR[GP1:91,1] = PR[GP1:90,1] + 72.227;
   1:  PR[GP1:91,2] = PR[GP1:90,2] + 100.094;
   1:L PR[91] 10mm/sec FINE;
   1:  PR[GP1:91,1] = PR[GP1:90,1] + 72.499;
